       //read cooling water temperature and flow variables 
       //-------------------------------------------------
       IF NOT "SY".SIM_ON THEN                                                                                        // K01: Spare
           "DIS".ACT_WTR_FLW_XT_SFT   := INT_TO_REAL(WORD_TO_INT("P_BM_ACT_WTR_FLW_XT_SFT":P))/100.0;      // K02: seed shaft
           "DIS".ACT_WTR_TMP_XT_SFT   := INT_TO_REAL(WORD_TO_INT("P_BM_ACT_WTR_TMP_XT_SFT":P))/40.0;       
           "DIS".ACT_WTR_FLW_GCH      := INT_TO_REAL(WORD_TO_INT("P_BM_ACT_WTR_FLW_GCH":P))/100.0;         // K03: gate chamber 
           "DIS".ACT_WTR_TMP_GCH      := INT_TO_REAL(WORD_TO_INT("P_BM_ACT_WTR_TMP_GCH":P))/40.0; 
           "DIS".ACT_WTR_FLW_GCH_H    := INT_TO_REAL(WORD_TO_INT("P_BM_ACT_WTR_FLW_GCH_H":P))/100.0;       // K04: gate chamber valve housing
           "DIS".ACT_WTR_TMP_GCH_H    := INT_TO_REAL(WORD_TO_INT("P_BM_ACT_WTR_TMP_GCH_H":P))/40.0;    
           "DIS".ACT_WTR_FLW_GCH_V    := INT_TO_REAL(WORD_TO_INT("P_BM_ACT_WTR_FLW_GCH_V":P))/100.0;       // K05: gate chamber valve
           "DIS".ACT_WTR_TMP_GCH_V    := INT_TO_REAL(WORD_TO_INT("P_BM_ACT_WTR_TMP_GCH_V":P))/40.0;    
           "DIS".ACT_WTR_FLW_VPTS     := INT_TO_REAL(WORD_TO_INT("P_BM_ACT_WTR_FLW_VPTS":P))/100.0;        // K06: view ports
           "DIS".ACT_WTR_TMP_VPTS     := INT_TO_REAL(WORD_TO_INT("P_BM_ACT_WTR_TMP_VPTS":P))/40.0;    
           "DIS".ACT_WTR_FLW_TCH      := INT_TO_REAL(WORD_TO_INT("P_BM_ACT_WTR_FLW_TCH":P))/100.0;         // K07: top chamber 
           "DIS".ACT_WTR_TMP_TCH      := INT_TO_REAL(WORD_TO_INT("P_BM_ACT_WTR_TMP_TCH":P))/40.0;    
           "DIS".ACT_WTR_FLW_TEC_FLG  := INT_TO_REAL(WORD_TO_INT("P_BM_ACT_WTR_FLW_TEC_FLG":P))/100.0;     // K08: technology flange
           "DIS".ACT_WTR_TMP_TEC_FLG  := INT_TO_REAL(WORD_TO_INT("P_BM_ACT_WTR_TMP_TEC_FLG":P))/40.0;    
                                                                                                   // K09: Spare
           "DIS".ACT_WTR_FLW_UP_FCH   := INT_TO_REAL(WORD_TO_INT("P_BM_ACT_WTR_FLW_UP_FCH":P))/100.0;      // K10: Upper furnace chamber
           "DIS".ACT_WTR_TMP_UP_FCH   := INT_TO_REAL(WORD_TO_INT("P_BM_ACT_WTR_TMP_UP_FCH":P))/40.0;    
           "DIS".ACT_WTR_FLW_FCH      := INT_TO_REAL(WORD_TO_INT("P_BM_ACT_WTR_FLW_FCH":P))/100.0;         // K11: Lower furnace chamber
           "DIS".ACT_WTR_TMP_FCH      := INT_TO_REAL(WORD_TO_INT("P_BM_ACT_WTR_TMP_FCH":P))/40.0;    
           "DIS".ACT_WTR_FLW_VSL      := INT_TO_REAL(WORD_TO_INT("P_BM_ACT_WTR_FLW_BCH":P))/100.0;         // K12: bottom chamber
           "DIS".ACT_WTR_TMP_VSL      := INT_TO_REAL(WORD_TO_INT("P_BM_ACT_WTR_TMP_BCH":P))/40.0;    
           "DIS".ACT_WTR_FLW_SOC_BCH  := INT_TO_REAL(WORD_TO_INT("P_BM_ACT_WTR_FLW_SOC_BCH":P))/100.0;     // K13: socket bottom chamber
           "DIS".ACT_WTR_TMP_SOC_BCH  := INT_TO_REAL(WORD_TO_INT("P_BM_ACT_WTR_TMP_SOC_BCH":P))/40.0;    
           "DIS".ACT_WTR_FLW_CUR_FEED := INT_TO_REAL(WORD_TO_INT("P_BM_ACT_WTR_FLW_CFT_M":P))/100.0;       // K14: current feed throught Main
           "DIS".ACT_WTR_TMP_CUR_FEED := INT_TO_REAL(WORD_TO_INT("P_BM_ACT_WTR_TMP_CFT_M":P))/40.0;    
           "DIS".ACT_WTR_FLW_CFT_2    := INT_TO_REAL(WORD_TO_INT("P_BM_ACT_WTR_FLW_CFT_B":P))/100.0;       // K15: current feed throughs Bottom
           "DIS".ACT_WTR_TMP_CFT_2    := INT_TO_REAL(WORD_TO_INT("P_BM_ACT_WTR_TMP_CFT_B":P))/40.0;    
         //DIS.ACT_WTR_FLW_ACC      := INT_TO_REAL(WORD_TO_INT(BM_ACT_WTR_FLW_ACC))/100.0;        // K16: Active cooling
         //DIS.ACT_WTR_TMP_ACC      := INT_TO_REAL(WORD_TO_INT(BM_ACT_WTR_TMP_ACC))/40.0;   
           "DIS".ACT_WTR_FLW_CR_SFT   := INT_TO_REAL(WORD_TO_INT("P_BM_ACT_WTR_FLW_CR_SFT":P))/100.0;      // K17: crucible shaft
           "DIS".ACT_WTR_TMP_CR_SFT   := INT_TO_REAL(WORD_TO_INT("P_BM_ACT_WTR_TMP_CR_SFT":P))/40.0;    
           "DIS".ACT_WTR_FLW_PWR_CAB  := INT_TO_REAL(WORD_TO_INT("P_BM_ACT_WTR_FLW_PWR_CAB":P))/100.0;     // K18: high current cables Main
           "DIS".ACT_WTR_TMP_PWR_CAB  := INT_TO_REAL(WORD_TO_INT("P_BM_ACT_WTR_TMP_PWR_CAB":P))/40.0;    
           "DIS".ACT_WTR_FLW_PWR_CAB2 := INT_TO_REAL(WORD_TO_INT("P_BM_ACT_WTR_FLW_PWR_CAB2":P))/100.0;    // K19: high current cables Bot
           "DIS".ACT_WTR_TMP_PWR_CAB2 := INT_TO_REAL(WORD_TO_INT("P_BM_ACT_WTR_TMP_PWR_CAB2":P))/40.0;    
           "DIS".ACT_WTR_FLW_HTR_1    := INT_TO_REAL(WORD_TO_INT("P_BM_ACT_WTR_FLW_HTR":P))/100.0;         // K20: heater power supply
           "DIS".ACT_WTR_TMP_HTR_1    := INT_TO_REAL(WORD_TO_INT("P_BM_ACT_WTR_TMP_HTR":P))/40.0;         
                                                                                                   // K21: Spare
                                                                                                   // K22: Spare
                                                                                                   // K23: Spare
           "DIS".ACT_WTR_FLW_GCH_ADDS      := INT_TO_REAL(WORD_TO_INT("P_BM_ACT_WTR_FLW_GCH_ADDS":P))/100.0;         // K24: gate chamber Additions
           "DIS".ACT_WTR_TMP_GCH_ADDS      := INT_TO_REAL(WORD_TO_INT(SHR(IN:= "P_BM_ACT_WTR_TMP_GCH_ADDS":P, N:= 2)))/10.0;    
         //DIS.ACT_WTR_FLW_PU       := INT_TO_REAL(WORD_TO_INT(BM_ACT_WTR_FLW_PU))/100.0;          // K25: pump unit
         //DIS.ACT_WTR_TMP_PU       := INT_TO_REAL(WORD_TO_INT(SHR(IN:= BM_ACT_WTR_TMP_PU, N:= 2)))/10.0;    
           "DIS".ACT_WTR_FLW_MAG_CO4  := INT_TO_REAL(WORD_TO_INT("P_BM_ACT_WTR_FLW_MAG_CO4":P))/100.0;     // K26: magnet compressor unit 4
           "DIS".ACT_WTR_TMP_MAG_CO4  := INT_TO_REAL(WORD_TO_INT(SHR(IN:= "P_BM_ACT_WTR_TMP_MAG_CO4":P, N:= 2)))/10.0;    
           "DIS".ACT_WTR_FLW_MAG_CO3  := INT_TO_REAL(WORD_TO_INT("P_BM_ACT_WTR_FLW_MAG_CO3":P))/100.0;     // K27: magnet compressor unit 3
           "DIS".ACT_WTR_TMP_MAG_CO3  := INT_TO_REAL(WORD_TO_INT(SHR(IN:= "P_BM_ACT_WTR_TMP_MAG_CO3":P, N:= 2)))/10.0;    
           "DIS".ACT_WTR_FLW_MAG_CO2  := INT_TO_REAL(WORD_TO_INT("P_BM_ACT_WTR_FLW_MAG_CO2":P))/100.0;     // K28: magnet compressor unit 2
           "DIS".ACT_WTR_TMP_MAG_CO2  := INT_TO_REAL(WORD_TO_INT(SHR(IN:= "P_BM_ACT_WTR_TMP_MAG_CO2":P, N:= 2)))/10.0;    
           "DIS".ACT_WTR_FLW_MAG_CO1  := INT_TO_REAL(WORD_TO_INT("P_BM_ACT_WTR_FLW_MAG_CO1":P))/100.0;     // K29: magnet compressor unit 1
           "DIS".ACT_WTR_TMP_MAG_CO1  := INT_TO_REAL(WORD_TO_INT(SHR(IN:= "P_BM_ACT_WTR_TMP_MAG_CO1":P, N:= 2)))/10.0;    
           "DIS".ACT_WTR_FLW_MAG_CAB  := INT_TO_REAL(WORD_TO_INT("P_BM_ACT_WTR_FLW_MAG_CAB":P))/100.0;     // K30: magnet power supply
           "DIS".ACT_WTR_TMP_MAG_CAB  := INT_TO_REAL(WORD_TO_INT(SHR(IN:= "P_BM_ACT_WTR_TMP_MAG_CAB":P, N:= 2)))/10.0;    

           "DIS".ACT_WTR_FLW_VAC_BYP  := INT_TO_REAL(WORD_TO_INT("P_BM_ACT_WTR_FLW_VAC_BYP":P))/100.0;     // Kxx: vacuum bypass tube
           "DIS".ACT_WTR_TMP_VAC_BYP  := INT_TO_REAL(WORD_TO_INT("P_BM_ACT_WTR_TMP_VAC_BYP":P))/40.0;  
       END_IF;


       //set water flow and temperature alarms
       //-------------------------------------
       "FLT".XT_TAS              :=  ("DIS".ACT_WTR_TMP_XT_SFT > "CNF".WTR_TMP_WRN);             // seed shaft
       "FLT".XT_WFS              :=  ("DIS".ACT_WTR_FLW_XT_SFT < "CNF".MIN_WTR_FLW_XT_SFT);       
       "FLT".WTR_TMP_GCH         :=  ("DIS".ACT_WTR_TMP_GCH > "CNF".WTR_TMP_WRN) OR              //gate chamber
                                   ("DIS".ACT_WTR_TMP_GCH_H > "CNF".WTR_TMP_WRN);              // gate chamber valve housing    
       "FLT".WTR_FLW_GCH         :=  ("DIS".ACT_WTR_FLW_GCH < "CNF".MIN_WTR_FLW_GCH) OR 
                                   ("DIS".ACT_WTR_FLW_GCH_H < "CNF".MIN_WTR_FLW_GCH_H);  
       "FLT".WTR_TMP_GCH_V       :=  ("DIS".ACT_WTR_TMP_GCH_V > "CNF".WTR_TMP_WRN);              //gate chamber valve
       "FLT".WTR_FLW_GCH_V       :=  ("DIS".ACT_WTR_FLW_GCH_V < "CNF".MIN_WTR_FLW_GCH_V); 
       "FLT".WTR_TMP_VPTS        :=  ("DIS".ACT_WTR_TMP_VPTS > "CNF".WTR_TMP_WRN);               //view ports
       "FLT".WTR_FLW_VPTS        :=  ("DIS".ACT_WTR_FLW_VPTS < "CNF".MIN_WTR_FLW_VPTS); 
       "FLT".WTR_TMP_TCH         :=  ("DIS".ACT_WTR_TMP_TCH > "CNF".WTR_TMP_WRN);                //top chamber
       "FLT".WTR_FLW_TCH         :=  ("DIS".ACT_WTR_FLW_TCH < "CNF".MIN_WTR_FLW_TCH);
       "FLT".WTR_TMP_TEC_FLG     :=  ("DIS".ACT_WTR_TMP_TEC_FLG > "CNF".WTR_TMP_WRN);            //technology flange
       "FLT".WTR_FLW_TEC_FLG     :=  ("DIS".ACT_WTR_FLW_TEC_FLG < "CNF".MIN_WTR_FLW_TEC_CHB);    
       "FLT".WTR_TMP_FCH         :=  ("DIS".ACT_WTR_TMP_UP_FCH > "CNF".WTR_TMP_WRN)OR            //upper furnace chamber
                                   ("DIS".ACT_WTR_TMP_FCH > "CNF".WTR_TMP_WRN);                //lower furnace chamber
       "FLT".WTR_FLW_FCH         :=  ("DIS".ACT_WTR_FLW_UP_FCH < "CNF".MIN_WTR_FLW_FCH)OR
                                   ("DIS".ACT_WTR_FLW_FCH < "CNF".MIN_WTR_FLW_FCH);
       "FLT".WTR_TMP_VSL         :=  ("DIS".ACT_WTR_TMP_VSL  > "CNF".WTR_TMP_WRN) OR             //bottom chamber
                                   ("DIS".ACT_WTR_TMP_SOC_BCH > "CNF".WTR_TMP_WRN);            //socket bottom chamber    
       "FLT".WTR_FLW_VSL         :=  ("DIS".ACT_WTR_FLW_VSL < "CNF".MIN_WTR_FLW_VSL) OR
                                   ("DIS".ACT_WTR_FLW_SOC_BCH < "CNF".MIN_WTR_FLW_VSL);    
       "FLT".WTR_TMP_CUR_FEED    :=  ("DIS".ACT_WTR_TMP_CUR_FEED > "CNF".WTR_TMP_WRN);           //current feed throughs heater 1
       "FLT".WTR_FLW_CUR_FEED    :=  ("DIS".ACT_WTR_FLW_CUR_FEED < "CNF".MIN_WTR_FLW_CUR_FEED); 
       "FLT".WTR_TMP_CFT_2       :=  ("DIS".ACT_WTR_TMP_CFT_2 > "CNF".WTR_TMP_WRN);              //current feed throughs heater 2
       "FLT".WTR_FLW_CFT_2       :=  ("DIS".ACT_WTR_FLW_CFT_2 < "CNF".MIN_WTR_FLW_CUR_FEED);
       "FLT".WTR_TMP_PWR_CAB     :=  ("DIS".ACT_WTR_TMP_PWR_CAB > "CNF".WTR_TMP_WRN)OR           //high current cables main
                                   ("DIS".ACT_WTR_TMP_PWR_CAB2 > "CNF".WTR_TMP_WRN);           //high current cables 2 bot    
       "FLT".WTR_FLW_PWR_CAB     :=  ("DIS".ACT_WTR_FLW_PWR_CAB < "CNF".MIN_WTR_FLW_PWR_CAB)OR 
                                   ("DIS".ACT_WTR_FLW_PWR_CAB2 < "CNF".MIN_WTR_FLW_PWR_CAB); 
       "FLT".WTR_TMP_CR_SFT      :=  ("DIS".ACT_WTR_TMP_CR_SFT > "CNF".WTR_TMP_WRN);             //crucible shaft
       "FLT".WTR_FLW_CR_SFT      :=  ("DIS".ACT_WTR_FLW_CR_SFT < "CNF".MIN_WTR_FLW_CR_SFT);    
       "FLT".WTR_TMP_HTR_1       :=  ("DIS".ACT_WTR_TMP_HTR_1 > "CNF".WTR_TMP_WRN);              //heater power supply
       IF "CNF".CONF_PWR_SPL_TYPE = 1 THEN 
          "FLT".WTR_FLW_HTR_1       :=  ("DIS".ACT_WTR_FLW_HTR_1 < "CNF".MIN_WTR_FLW_PWR_HTR_1); 
       END_IF;
       IF "CNF".CONF_PWR_SPL_TYPE = 2 THEN 
          "FLT".WTR_FLW_HTR_1       :=  ("DIS".ACT_WTR_FLW_HTR_1 < "CNF".MIN_WTR_FLW_INJ_HTR_1); 
       END_IF;
     //FLT.WTR_TMP_ACC         :=  (DIS.ACT_WTR_TMP_ACC > CNF.WTR_TMP_WRN);                 // active cooling
     //FLT.WTR_FLW_ACC         :=  (DIS.ACT_WTR_FLW_ACC < CNF.MIN_WTR_FLW_ACC_IN);         
       "FLT".WTR_TMP_GCH_ADDS         :=  ("DIS".ACT_WTR_TMP_GCH_ADDS > "CNF".WTR_TMP_WRN);                 // chamber parts, view ports
       "FLT".WTR_FLW_GCH_ADDS         :=  ("DIS".ACT_WTR_FLW_GCH_ADDS < "CNF".MIN_WTR_FLW_GCH_ADDS);    

       "FLT".MAG_TAS             :=  ("DIS".ACT_WTR_TMP_MAG_CO1 > "CNF".WTR_TMP_WRN) OR           // magnet compressor unit 1
                                   ("DIS".ACT_WTR_TMP_MAG_CO2 > "CNF".WTR_TMP_WRN) OR           // magnet compressor unit 2
                                   ("DIS".ACT_WTR_TMP_MAG_CO3 > "CNF".WTR_TMP_WRN) OR           // magnet compressor unit 3
                                   ("DIS".ACT_WTR_TMP_MAG_CO4 > "CNF".WTR_TMP_WRN) OR           // magnet compressor unit 4
                                   ("DIS".ACT_WTR_TMP_MAG_CAB > "CNF".WTR_TMP_WRN);             // magnet power supply
       "FLT".MAG_WFS             :=  ("DIS".ACT_WTR_FLW_MAG_CO1 < "CNF".MIN_WTR_FLW_MAG_COMP) OR    
                                   ("DIS".ACT_WTR_FLW_MAG_CO2 < "CNF".MIN_WTR_FLW_MAG_COMP) OR    
                                   ("DIS".ACT_WTR_FLW_MAG_CO3 < "CNF".MIN_WTR_FLW_MAG_COMP) OR    
                                   ("DIS".ACT_WTR_FLW_MAG_CO4 < "CNF".MIN_WTR_FLW_MAG_COMP) OR    
                                   ("DIS".ACT_WTR_FLW_MAG_CAB < "CNF".MIN_WTR_FLW_MAG_CAB);    

       "FLT".WTR_TMP_VAC_BYP     :=  ("DIS".ACT_WTR_TMP_VAC_BYP > "CNF".WTR_TMP_WRN);                // vacuum bypass tube - not included in interlocks
       "FLT".WTR_FLW_VAC_BYP     :=  ("DIS".ACT_WTR_FLW_VAC_BYP < "CNF".MIN_WTR_FLW_VAC_BYP);

       //built shut down flag low water flow (current feed throughs heater 2 not included)
       //---------------------------------------------------------------------------------
       #low_wtr_flw :=      "FLT".XT_WFS OR                   //seed shaft
                           "FLT".WTR_FLW_GCH OR              //gate chamber or gate chamber valve housing
                           "FLT".WTR_FLW_GCH_V OR            //gate chamber valve
                           "FLT".WTR_FLW_VPTS OR             //view ports
                           "FLT".WTR_FLW_TCH OR              //top chamber
                           "FLT".WTR_FLW_TEC_FLG OR          //technology flange
                           "FLT".WTR_FLW_FCH OR              //upper furnace chamber or lower furnace chamber
                           "FLT".WTR_FLW_VSL OR              //bottom chamber or socket bottom chamber
                           "FLT".WTR_FLW_CR_SFT OR           //crucible shaft
                           "FLT".WTR_FLW_HTR_1 OR            //heater power supply
                           "FLT".WTR_FLW_GCH_ADDS;           //gate chamber additions

       //built shut down flag low water flow heater 1(only current feed throughs and cables of heater 1)
       //-----------------------------------------------------------------------------------------------
       #low_wtr_flw_htr_1   :=  ("DIS".ACT_WTR_FLW_CUR_FEED < "CNF".MIN_WTR_FLW_CUR_FEED) OR        //current feed throughs heater 1
                               "DIS".ACT_WTR_FLW_PWR_CAB < "CNF".MIN_WTR_FLW_PWR_CAB;             //high current cables heater 1

       //built shut down flag low water flow heater 2(only current feed throughs and cables of heater 2)
       //-----------------------------------------------------------------------------------------------
       #low_wtr_flw_htr_2   :=  ("DIS".ACT_WTR_FLW_CFT_2 < "CNF".MIN_WTR_FLW_CUR_FEED) OR           //current feed throughs heater 2
                               "DIS".ACT_WTR_FLW_PWR_CAB2 < "CNF".MIN_WTR_FLW_PWR_CAB;             //high current cables heater 2

       //built shut down flag high water temperature (current feed throughs heater 2 not included)
       //-----------------------------------------------------------------------------------------
       #high_wtr_tmp    :=  ("DIS".ACT_WTR_TMP_XT_SFT > "CNF".MAX_WTR_TMP_LIM)OR    //seed shaft
                           ("DIS".ACT_WTR_TMP_GCH > "CNF".MAX_WTR_TMP_LIM) OR      //gate chamber
                           ("DIS".ACT_WTR_TMP_GCH_H > "CNF".MAX_WTR_TMP_LIM)OR     //gate chamber valve housing    
                           ("DIS".ACT_WTR_TMP_GCH_V > "CNF".MAX_WTR_TMP_LIM)OR     //gate chamber valve
                           ("DIS".ACT_WTR_TMP_VPTS > "CNF".MAX_WTR_TMP_LIM)OR      //view ports
                           ("DIS".ACT_WTR_TMP_TCH > "CNF".MAX_WTR_TMP_LIM)OR       //top chamber
                           ("DIS".ACT_WTR_TMP_TEC_FLG > "CNF".MAX_WTR_TMP_LIM)OR   //technology flange
                           ("DIS".ACT_WTR_TMP_UP_FCH > "CNF".MAX_WTR_TMP_LIM)OR    //upper furnace chamber
                           ("DIS".ACT_WTR_TMP_FCH > "CNF".MAX_WTR_TMP_LIM)OR       //lower furnace chamber
                           ("DIS".ACT_WTR_TMP_VSL  > "CNF".MAX_WTR_TMP_LIM) OR     //bottom chamber
                           ("DIS".ACT_WTR_TMP_SOC_BCH > "CNF".MAX_WTR_TMP_LIM)OR   //socket bottom chamber    
                           ("DIS".ACT_WTR_TMP_CR_SFT > "CNF".MAX_WTR_TMP_LIM)OR    //crucible shaft
                           ("DIS".ACT_WTR_TMP_HTR_1 > "CNF".MAX_WTR_TMP_LIM)OR     //heater power supply
                           ("DIS".ACT_WTR_TMP_GCH_ADDS > "CNF".MAX_WTR_TMP_LIM);   //gate chamber additions

       "FLT".WTR_TMP_VAC_BYP     :=  ("DIS".ACT_WTR_TMP_VAC_BYP > "CNF".WTR_TMP_WRN);                // vacuum bypass tube - not included in interlocks
       "FLT".WTR_FLW_VAC_BYP     :=  ("DIS".ACT_WTR_FLW_VAC_BYP < "CNF".MIN_WTR_FLW_VAC_BYP);

       //built shut down flag high cooling water temperature heater 1
       //------------------------------------------------------------
       #high_wtr_tmp_htr_1  :=  ("DIS".ACT_WTR_TMP_CUR_FEED > "CNF".MAX_WTR_TMP_LIM) OR //current feed throughs heater 1
                               ("DIS".ACT_WTR_TMP_PWR_CAB > "CNF".MAX_WTR_TMP_LIM);    //high current cables heater 1

       //built shut down flag high cooling water temperature heater 2
       //------------------------------------------------------------
       #high_wtr_tmp_htr_2  :=  ("DIS".ACT_WTR_TMP_CFT_2 > "CNF".MAX_WTR_TMP_LIM) OR    //current feed throughs heater 2
                               ("DIS".ACT_WTR_TMP_PWR_CAB2 > "CNF".MAX_WTR_TMP_LIM);   //high current cables heater 2

       //set alarm high water temperature
       //--------------------------------            
       "FLT".WTR_TMP_HIGH_LIM    :=  #high_wtr_tmp OR            
                                   #high_wtr_tmp_htr_1 OR
                                   #high_wtr_tmp_htr_2;

       //reconnect heater 1 after power fail
       //-----------------------------------
       IF "DV".PWR_FAIL_HTR_1_ON THEN
           "KYA".SET_HTR_1_PWR := "AV".PWR_FAIL_HTR_1_PWR;      // restore last power value

           IF ("LT".HTR_1_ON) THEN  //AND PDO.HTR_1_ENB
               "DV".PWR_FAIL_HTR_1_ON := false;               // delete request, if heater on
               "AV".PWR_FAIL_HTR_1_PWR := 0.0;
           END_IF;
       END_IF;

       //check heater power supply interlocks affecting all heater
       //---------------------------------------------------------
       #htr_itl_ok      :=  "BM_HTR_ITL" (aps             :=      NOT "PDI".FCH_APS,  
                                       tas             :=      NOT #high_wtr_tmp,
                                       on_dly_tas      :=      "HTR_TAS_DLY", 
                                       dly_time_tas    :=      T#30s,
                                       wfs             :=      NOT #low_wtr_flw,
                                       on_dly_wfs      :=      "HTR_WFS_DLY", 
                                       dly_time_wfs    :=      T#30s,                                               
                                       aux             :=      "DV".MAIN_SWITCH_ON AND
                                                              ("PDI".ACC_SC_HTR_OK AND   //ACC heater safety circuit
                                                               "PDI".ACC_SC_WTR_OK OR    //ACC water safety circuit
                                                               NOT "DV".ACC_INST),           //ACC installed?
                                       on_dly_aux      :=      "HTR_AUX_DLY", 
                                       dly_time_aux    :=      T#1s);  

       //extend reset flag earth fault detection
       //---------------------------------------   
       "LT".RESET_ERR_HTR_ETH    := "SysOffdelay" (DIN     := "KYD".RESET_ERR_HTR_ETH,
                                               SetTime := 20,                          // setp. time
                                               ActTime := #rst_err_htr_eth_dly,         // act. time
                                               Tick    := "SysTick100ms");               // timebase (100ms)


       //TLU switching power supply
       //--------------------------
       //check heater 1 interlock
       //------------------------
       #htr_1_itl_ok    :=  "BM_HTR_ITL" (aps             :=      true,  
                                       tas             :=      NOT #high_wtr_tmp_htr_1,
                                       on_dly_tas      :=      "HTR_1_TAS_DLY", 
                                       dly_time_tas    :=      T#30s,
                                       wfs             :=      NOT #low_wtr_flw_htr_1,
                                       on_dly_wfs      :=      "HTR_1_WFS_DLY", 
                                       dly_time_wfs    :=      T#30s,                                               
                                       aux             :=      NOT "FLT".HTR_1_PWR_SPL,
                                       on_dly_aux      :=      "HTR_1_AUX_DLY", 
                                       dly_time_aux    :=      T#1s);                                

       //check heater 2 interlock
       //------------------------
       #htr_2_itl_ok    :=  "BM_HTR_ITL" (aps             :=      true,  
                                       tas             :=      NOT #high_wtr_tmp_htr_2,
                                       on_dly_tas      :=      "HTR_2_TAS_DLY", 
                                       dly_time_tas    :=      T#30s,
                                       wfs             :=      NOT #low_wtr_flw_htr_2,
                                       on_dly_wfs      :=      "HTR_2_WFS_DLY", 
                                       dly_time_wfs    :=      T#30s,                                               
                                       aux             :=      NOT "FLT".HTR_2_PWR_SPL,
                                       on_dly_aux      :=      "HTR_2_AUX_DLY", 
                                       dly_time_aux    :=      T#1s);                                

       //call control module of heater 1
       //-------------------------------
       "CM_ITL_IO"(ADR := 30,
              KYD_ON := ("KYD".HTR_1_ON AND NOT "DV".EMG_DRV_ENB) OR "DV".PWR_FAIL_HTR_1_ON,
              KYD_OFF:= "KYD".HTR_1_OFF OR "DV".PWR_FAIL_HTR_OFF OR "DV".EMG_DVC_OFF,
              AUTO := "APC".AUTOMATIC,
              DC_ON:= "DC".HTR_1_ON,
              CON1 := "PDI".EMO,
              CON2 := "DV".MAIN_SWITCH_ON,
              CON3 := #htr_itl_ok,
              CON4 := #htr_1_itl_ok,               
              CON5 := "SysLog1",
              CON6 := "SysLog1",                             
              CON7 := "SysLog1",                             
              CON8 := "SysLog1",
              ITL_OUT:= "STA_ITL_CAUSE",
              LT_OUT := "LT".HTR_1_ON);

       //set power enable delayed
       //------------------------
       #htr_1_enb     := "SysOndelay"(DIN     := "LT".HTR_1_ON,
                                   SetTime := 10,                // 1 sec. delay after power on
                                   ActTime := #htr_1_pwr_enb_dly, // act. time
                                   Tick    := "SysTick100ms");     // timebase (100ms)

       //heater supply power on
       //----------------------
       "PDO".HTR_PWR_ON    :=  "LT".HTR_1_ON;               

       //reset power set point if heater enable is gone
       //----------------------------------------------
       IF NOT #htr_1_enb  THEN
           "KYA".SET_HTR_1_PWR  := 0.0;
           "CTL".SET_HTR_1_PWR  := 0.0;
       END_IF;

       //extent reset flag
       //-----------------
       "LT".RST_HTR_1_PWR_SPL := "SysOffdelay"(DIN     := "KYD".RST_HTR_1_PWR_SPL,
                                           SetTime := 20,                          // setp. time
                                           ActTime := #rst_htr_1_pwr_spl_dly,       // act. time
                                           Tick    := "SysTick100ms");               // timebase (100ms)

       //call control module of heater 2
       //-------------------------------
       "CM_ITL_IO"(ADR := 31,
              KYD_ON := ("KYD".HTR_2_ON AND NOT "DV".EMG_DRV_ENB) OR "DV".PWR_FAIL_HTR_2_ON,
              KYD_OFF:= "KYD".HTR_2_OFF OR "DV".PWR_FAIL_HTR_OFF OR "DV".EMG_DVC_OFF,
              AUTO := "APC".AUTOMATIC,
              DC_ON:= "DC".HTR_2_ON,
              CON1 := "PDI".EMO,
              CON2 := "DV".MAIN_SWITCH_ON,
              CON3 := #htr_itl_ok,
              CON4 := #htr_2_itl_ok,               
              CON5 := "SysLog1",
              CON6 := "SysLog1",                             
              CON7 := "SysLog1",                             
              CON8 := "SysLog1",
              ITL_OUT:= "STA_ITL_CAUSE",
              LT_OUT := "LT".HTR_2_ON);

       //set power enable delayed
       //------------------------
       #htr_2_enb     := "SysOndelay"(DIN     := "LT".HTR_2_ON,
                                   SetTime := 10,                // 1 sec. delay after power on
                                   ActTime := #htr_2_pwr_enb_dly, // act. time
                                   Tick    := "SysTick100ms");     // timebase (100ms)

       //set output heater 2 (used in ekz_sm_pwr_fail)
       //---------------------------------------------
      // PDO.HTR_2_ON    :=  LT.HTR_2_ON;               

       //reset power set point if heater enable is gone
       //----------------------------------------------
       IF NOT #htr_2_enb  THEN
           "KYA".SET_HTR_2_PWR  := 0.0;
           "CTL".SET_HTR_2_PWR  := 0.0;
       END_IF;

       //extent reset flag
       //-----------------
       "LT".RST_HTR_2_PWR_SPL := "SysOffdelay"(DIN     := "KYD".RST_HTR_2_PWR_SPL,
                                           SetTime := 20,                          // setp. time
                                           ActTime := #rst_htr_2_pwr_spl_dly,       // act. time
                                           Tick    := "SysTick100ms");               // timebase (100ms)


       //call communication module with TLU profibus interface
       //-----------------------------------------------------
       IF "CNF".CONF_PWR_SPL_TYPE = 1 THEN    
           //delay communication 
           //-------------------
           #start_htr_com := "SysOndelay"(DIN     := "PDO".HTR_PWR_ON,
                                       SetTime := 30,                  // setp. time
                                       ActTime := #com_heater_dly,      // act. time
                                       Tick    := "SysTick100ms");

           IF #start_htr_com THEN 

               #PM_TLU_HTR_1(   htr_enb         :=  #htr_1_enb, 
                               htr_rst         :=  "LT".RST_HTR_1_PWR_SPL,
                               fst_byte_offs   :=  0,        
                               dp_adress       :=  16#380,                 //addr: 896      
                               set_htr_pwr     :=  "CTL".SET_HTR_1_PWR,
                               htr_pwr_rng     :=  "CNF".HTR_1_PWR_RANGE,
                               htr_cur_rng     :=  "CNF".HTR_1_CUR_RANGE,
                               htr_vlt_rng     :=  "CNF".HTR_1_VLT_RANGE);
           END_IF;                

           "AV".ACT_HTR_1_PWR        :=  #PM_TLU_HTR_1.act_htr_pwr; 
           "AV".ACT_HTR_1_CUR        :=  #PM_TLU_HTR_1.act_htr_cur; 
           "AV".ACT_HTR_1_VLT        :=  #PM_TLU_HTR_1.act_htr_vlt; 

           "FLT".HTR_1_PWR_SPL_WRN   :=  #PM_TLU_HTR_1.sta_warn;  
           "FLT".HTR_1_PWR_SPL       :=  #PM_TLU_HTR_1.sta_error;  

           #htr_1_is_on             :=  #PM_TLU_HTR_1.sta_htr_on;         
           #htr_1_pi_mode           :=  #PM_TLU_HTR_1.sta_pi_mode;     
           #htr_1_pu_mode           :=  #PM_TLU_HTR_1.sta_pu_mode;      
           #htr_1_i_mode            :=  #PM_TLU_HTR_1.sta_i_mode;       
           #htr_1_u_mode            :=  #PM_TLU_HTR_1.sta_u_mode;       
           #htr_1_sta_saved         :=  #PM_TLU_HTR_1.sta_saved;         
           #htr_1_flt_i_pri         :=  #PM_TLU_HTR_1.flt_i_pri;       
           #htr_1_flt_i_max         :=  #PM_TLU_HTR_1.flt_i_max;        
           #htr_1_flt_u_max         :=  #PM_TLU_HTR_1.flt_u_max;        
           #htr_1_flt_wire          :=  #PM_TLU_HTR_1.flt_wire;           
           #htr_1_flt_flash         :=  #PM_TLU_HTR_1.flt_flash;          
           #htr_1_flt_trafo         :=  #PM_TLU_HTR_1.flt_trafo;         
           #htr_1_flt_data_flow     :=  #PM_TLU_HTR_1.flt_data_flow;    
           #htr_1_flt_data_com      :=  #PM_TLU_HTR_1.flt_data_com;      
           #htr_1_flt_data          :=  #PM_TLU_HTR_1.flt_data;       
           #htr_1_flt_tast          :=  #PM_TLU_HTR_1.flt_tast;            
           #htr_1_flt_ua_max        :=  #PM_TLU_HTR_1.flt_ua_max;          
           #htr_1_flt_u_min         :=  #PM_TLU_HTR_1.flt_u_min;          
           #htr_1_flt_temp          :=  #PM_TLU_HTR_1.flt_temp;            
           #htr_1_flt_sense         :=  #PM_TLU_HTR_1.flt_sense;         
           #htr_1_flt_igbt          :=  #PM_TLU_HTR_1.flt_igbt;          
           #htr_1_flt_dioden        :=  #PM_TLU_HTR_1.flt_dioden;       
           #htr_1_flt_3             :=  #PM_TLU_HTR_1.flt_3;             
           #htr_1_flt_shunt         :=  #PM_TLU_HTR_1.flt_shunt;         
           #htr_1_flt_board         :=  #PM_TLU_HTR_1.flt_board;         
           #htr_1_flt_6             :=  #PM_TLU_HTR_1.flt_6;            
           #htr_1_flt_soft          :=  #PM_TLU_HTR_1.flt_soft;          
           #htr_1_flt_timeout       :=  #PM_TLU_HTR_1.flt_timeout;        
           #htr_1_flt_short         :=  #PM_TLU_HTR_1.flt_short;    

           //errors heater 1 earthing monitoring
           //------------------ 
           IF  (("P_BM_HTR_1_ETH_STA":P AND 2#0001_0000) = 2#0001_0000) THEN  
               #flt_htr_1_eth_range := true;     //range error
           ELSE     
               #flt_htr_1_eth_range := false;
           END_IF;

           IF (("P_BM_HTR_1_ETH_STA":P AND 2#0010_0000) = 2#0010_0000) THEN 
               #flt_htr_1_eth_hw := true;       //intern hardware error
           ELSE     
               #flt_htr_1_eth_hw := false;
           END_IF;

           IF (("P_BM_HTR_1_ETH_STA":P AND 2#0100000) = 2#0100_0000) THEN 
               #flt_htr_1_eth_bus := true;      //bus error
           ELSE     
               #flt_htr_1_eth_bus := false;
           END_IF;

           //heater 2
           //--------  
           IF #start_htr_com THEN 

               #PM_TLU_HTR_2(   htr_enb         :=  #htr_2_enb, 
                               htr_rst         :=  "LT".RST_HTR_2_PWR_SPL,
                               fst_byte_offs   :=  0,        
                               dp_adress       :=  16#3C0,                 //addr: 960      
                               set_htr_pwr     :=  "CTL".SET_HTR_2_PWR,
                               htr_pwr_rng     :=  "CNF".HTR_2_PWR_RANGE,
                               htr_cur_rng     :=  "CNF".HTR_2_CUR_RANGE,
                               htr_vlt_rng     :=  "CNF".HTR_2_VLT_RANGE);
           END_IF;                

           "AV".ACT_HTR_2_PWR        :=  #PM_TLU_HTR_2.act_htr_pwr; 
           "AV".ACT_HTR_2_CUR        :=  #PM_TLU_HTR_2.act_htr_cur; 
           "AV".ACT_HTR_2_VLT        :=  #PM_TLU_HTR_2.act_htr_vlt; 

           "FLT".HTR_2_PWR_SPL_WRN   :=  #PM_TLU_HTR_2.sta_warn;  
           "FLT".HTR_2_PWR_SPL       :=  #PM_TLU_HTR_2.sta_error;    

           #htr_2_is_on             :=  #PM_TLU_HTR_2.sta_htr_on;         
           #htr_2_pi_mode           :=  #PM_TLU_HTR_2.sta_pi_mode;     
           #htr_2_pu_mode           :=  #PM_TLU_HTR_2.sta_pu_mode;      
           #htr_2_i_mode            :=  #PM_TLU_HTR_2.sta_i_mode;       
           #htr_2_u_mode            :=  #PM_TLU_HTR_2.sta_u_mode;       
           #htr_2_sta_saved         :=  #PM_TLU_HTR_2.sta_saved;         
           #htr_2_flt_i_pri         :=  #PM_TLU_HTR_2.flt_i_pri;       
           #htr_2_flt_i_max         :=  #PM_TLU_HTR_2.flt_i_max;        
           #htr_2_flt_u_max         :=  #PM_TLU_HTR_2.flt_u_max;        
           #htr_2_flt_wire          :=  #PM_TLU_HTR_2.flt_wire;           
           #htr_2_flt_flash         :=  #PM_TLU_HTR_2.flt_flash;          
           #htr_2_flt_trafo         :=  #PM_TLU_HTR_2.flt_trafo;         
           #htr_2_flt_data_flow     :=  #PM_TLU_HTR_2.flt_data_flow;    
           #htr_2_flt_data_com      :=  #PM_TLU_HTR_2.flt_data_com;      
           #htr_2_flt_data          :=  #PM_TLU_HTR_2.flt_data;       
           #htr_2_flt_tast          :=  #PM_TLU_HTR_2.flt_tast;            
           #htr_2_flt_ua_max        :=  #PM_TLU_HTR_2.flt_ua_max;          
           #htr_2_flt_u_min         :=  #PM_TLU_HTR_2.flt_u_min;          
           #htr_2_flt_temp          :=  #PM_TLU_HTR_2.flt_temp;            
           #htr_2_flt_sense         :=  #PM_TLU_HTR_2.flt_sense;         
           #htr_2_flt_igbt          :=  #PM_TLU_HTR_2.flt_igbt;          
           #htr_2_flt_dioden        :=  #PM_TLU_HTR_2.flt_dioden;       
           #htr_2_flt_3             :=  #PM_TLU_HTR_2.flt_3;             
           #htr_2_flt_shunt         :=  #PM_TLU_HTR_2.flt_shunt;         
           #htr_2_flt_board         :=  #PM_TLU_HTR_2.flt_board;         
           #htr_2_flt_6             :=  #PM_TLU_HTR_2.flt_6;            
           #htr_2_flt_soft          :=  #PM_TLU_HTR_2.flt_soft;          
           #htr_2_flt_timeout       :=  #PM_TLU_HTR_2.flt_timeout;        
           #htr_2_flt_short         :=  #PM_TLU_HTR_2.flt_short;  

           //errors heater 2 earthing monitoring
           //------------------ 
           IF  (("P_BM_HTR_2_ETH_STA":P AND 2#0001_0000) = 2#0001_0000) THEN  
               #flt_htr_2_eth_range := true;    //range error
           ELSE     
               #flt_htr_2_eth_range := false;
           END_IF;

           IF (("P_BM_HTR_2_ETH_STA":P AND 2#0010_0000) = 2#0010_0000) THEN 
               #flt_htr_2_eth_hw := true;       //intern hardware error
           ELSE     
               #flt_htr_2_eth_hw := false;
           END_IF;

           IF (("P_BM_HTR_2_ETH_STA":P AND 2#0100000) = 2#0100_0000) THEN 
               #flt_htr_2_eth_bus := true;      //bus error
           ELSE     
               #flt_htr_2_eth_bus := false;
           END_IF;

           // heater earthing monitoring error on HMI
           //------------------
           "FLT".HTR_ERH_COMM :=   #flt_htr_1_eth_range 
                              OR #flt_htr_1_eth_hw 
                              OR #flt_htr_1_eth_bus 
                              OR #flt_htr_2_eth_range
                              OR #flt_htr_2_eth_hw
                              OR #flt_htr_2_eth_bus;

           // reset heater earthing monitoring errors
           //------------------ 
           IF  "LT".RESET_ERR_HTR_ETH THEN 
               "P_BM_HTR_1_ETH_CTRL":P := 2#0100_0000;
               "P_BM_HTR_2_ETH_CTRL":P := 2#0100_0000;
           ELSE
               "P_BM_HTR_1_ETH_CTRL":P := 2#0000_0000;
               "P_BM_HTR_2_ETH_CTRL":P := 2#0000_0000;
           END_IF;

       END_IF;

       IF "CNF".CONF_PWR_SPL_TYPE = 2 THEN
           //call communication module with Injet profinet interface
           //-----------------------------------------------------
           //call Injet function  
           #PM_INJET_HTR     (htr_1_enb     := #htr_1_enb,  
                             htr_2_enb     := #htr_2_enb,     
                             set_htr_1_pwr := "CTL".SET_HTR_1_PWR,
                             set_htr_2_pwr := "CTL".SET_HTR_2_PWR);

           //heater 1 actual value                   
           "AV".ACT_HTR_1_PWR           :=  #PM_INJET_HTR.htr_1_act_pwr; 
           "AV".ACT_HTR_1_CUR           :=  #PM_INJET_HTR.htr_1_act_cur; 
           "AV".ACT_HTR_1_VLT           :=  #PM_INJET_HTR.htr_1_act_vlt;
           "DIS".ACT_HTR1_ETH_VLT_PLUS  :=  #PM_INJET_HTR.htr_1_eth_vlt_plus;   // Erdschluss黚erwachung 
           "DIS".ACT_HTR1_ETH_VLT_MINUS :=  #PM_INJET_HTR.htr_1_eth_vlt_minus;  

           "FLT".HTR1_COMM_ERR       :=  #PM_INJET_HTR.htr_1_flt_comm;
           "FLT".HTR2_COMM_ERR       :=  #PM_INJET_HTR.htr_2_flt_comm;  
           "FLT".HTR1_RCT_TMP        :=  #PM_INJET_HTR.flt_htr1_rct_tmp; // temperature monitoring for heater 1 power supply filter reactor, limit by 85癈

           "FLT".HTR1_RCT_TMP        :=  #PM_INJET_HTR.flt_htr2_rct_tmp; // temperature monitoring for heater 2 power supply filter reactor, limit by 85癈

           "FLT".PWR_SPL_APF_ERR     :=  #PM_INJET_HTR.flt_pwr_spl_APF;
           "FLT".PWR_SPL_CTL_ERR     :=  #PM_INJET_HTR.htr_1_flt_ctrl OR #PM_INJET_HTR.htr_2_flt_ctrl;// 
           "FLT".HTR_1_ETH           :=  #PM_INJET_HTR.htr_1_flt_erd_plus OR #PM_INJET_HTR.htr_1_flt_erd_min;
           "FLT".HTR_2_ETH           :=  #PM_INJET_HTR.htr_2_flt_erd_plus OR #PM_INJET_HTR.htr_2_flt_erd_min;

           "AV".ACT_HTR_2_PWR           :=  #PM_INJET_HTR.htr_2_act_pwr; 
           "AV".ACT_HTR_2_CUR           :=  #PM_INJET_HTR.htr_2_act_cur; 
           "AV".ACT_HTR_2_VLT           :=  #PM_INJET_HTR.htr_2_act_vlt;
           "DIS".ACT_HTR2_ETH_VLT_PLUS  :=  #PM_INJET_HTR.htr_2_eth_vlt_plus;   // Erdschluss黚erwachung 
           "DIS".ACT_HTR2_ETH_VLT_MINUS :=  #PM_INJET_HTR.htr_2_eth_vlt_minus;  


           #flt_pwr_spl_panel_comm  := #PM_INJET_HTR.flt_pwr_spl_panel_comm;
           #htr_1_remote            := #PM_INJET_HTR.htr_1_remote;
           #comm_ok                 := #PM_INJET_HTR.comm_ok;
           #htr_pwr_spl_cool_wtr_flt:= #PM_INJET_HTR.htr_pwr_spl_cool_wtr_flt;
           #htr_pwr_spl_cool_wtr_wrn:= #PM_INJET_HTR.htr_pwr_spl_cool_wtr_wrn;


           #htr_1_flt_save          := #PM_INJET_HTR.htr_1_flt_save;
           #htr_1_flt_ac_pha        := #PM_INJET_HTR.htr_1_flt_ac_pha;
           #htr_1_flt_tmp           := #PM_INJET_HTR.htr_1_flt_tmp;
           #htr_1_flt_cur           := #PM_INJET_HTR.htr_1_flt_cur;
           #htr_1_flt_cool_wtr      := #PM_INJET_HTR.htr_1_flt_cool_wtr;
           #htr_1_flt_term          := #PM_INJET_HTR.htr_1_flt_term;
           #htr_1_mod1_flt_syn_kab := #PM_INJET_HTR.htr_1_mod1_flt_syn_kab;
           #htr_1_mod1_flt_sys_tmp := #PM_INJET_HTR.htr_1_mod1_flt_sys_tmp;
           #htr_1_mod1_flt_drv     := #PM_INJET_HTR.htr_1_mod1_flt_drv;
           #htr_1_mod1_flt_cur     := #PM_INJET_HTR.htr_1_mod1_flt_cur;
           #htr_1_mod1_flt_vlt     := #PM_INJET_HTR.htr_1_mod1_flt_vlt;
           #htr_1_mod1_flt_save    := #PM_INJET_HTR.htr_1_mod1_flt_save;
           #htr_1_mod1_flt_rect    := #PM_INJET_HTR.htr_1_mod1_flt_rect;
           #htr_1_mod1_flt_tmp     := #PM_INJET_HTR.htr_1_mod1_flt_tmp;


           #htr_1_mod2_flt_syn_kab := #PM_INJET_HTR.htr_1_mod2_flt_syn_kab;
           #htr_1_mod2_flt_sys_tmp := #PM_INJET_HTR.htr_1_mod2_flt_sys_tmp;
           #htr_1_mod2_flt_drv     := #PM_INJET_HTR.htr_1_mod2_flt_drv;
           #htr_1_mod2_flt_cur     := #PM_INJET_HTR.htr_1_mod2_flt_cur;
           #htr_1_mod2_flt_vlt     := #PM_INJET_HTR.htr_1_mod2_flt_vlt;
           #htr_1_mod2_flt_save    := #PM_INJET_HTR.htr_1_mod2_flt_save;
           #htr_1_mod2_flt_rect    := #PM_INJET_HTR.htr_1_mod2_flt_rect;
           #htr_1_mod2_flt_tmp     := #PM_INJET_HTR.htr_1_mod2_flt_tmp;


           #htr_1_mod3_flt_syn_kab := #PM_INJET_HTR.htr_1_mod3_flt_syn_kab;
           #htr_1_mod3_flt_sys_tmp := #PM_INJET_HTR.htr_1_mod3_flt_sys_tmp;
           #htr_1_mod3_flt_drv     := #PM_INJET_HTR.htr_1_mod3_flt_drv;
           #htr_1_mod3_flt_cur     := #PM_INJET_HTR.htr_1_mod3_flt_cur;
           #htr_1_mod3_flt_vlt     := #PM_INJET_HTR.htr_1_mod3_flt_vlt;
           #htr_1_mod3_flt_save    := #PM_INJET_HTR.htr_1_mod3_flt_save;
           #htr_1_mod3_flt_rect    := #PM_INJET_HTR.htr_1_mod3_flt_rect;
           #htr_1_mod3_flt_tmp     := #PM_INJET_HTR.htr_1_mod3_flt_tmp;

           #htr_1_mod4_flt_syn_kab := #PM_INJET_HTR.htr_1_mod4_flt_syn_kab;
           #htr_1_mod4_flt_sys_tmp := #PM_INJET_HTR.htr_1_mod4_flt_sys_tmp;
           #htr_1_mod4_flt_drv     := #PM_INJET_HTR.htr_1_mod4_flt_drv;
           #htr_1_mod4_flt_cur     := #PM_INJET_HTR.htr_1_mod4_flt_cur;
           #htr_1_mod4_flt_vlt     := #PM_INJET_HTR.htr_1_mod4_flt_vlt;
           #htr_1_mod4_flt_save    := #PM_INJET_HTR.htr_1_mod4_flt_save;
           #htr_1_mod4_flt_rect    := #PM_INJET_HTR.htr_1_mod4_flt_rect;
           #htr_1_mod4_flt_tmp     := #PM_INJET_HTR.htr_1_mod4_flt_tmp;  

           #htr_2_remote           := #PM_INJET_HTR.htr_2_remote;
           #htr_2_flt_save         := #PM_INJET_HTR.htr_2_flt_save;
           #htr_2_flt_ac_pha       := #PM_INJET_HTR.htr_2_flt_ac_pha;
           #htr_2_flt_tmp          := #PM_INJET_HTR.htr_2_flt_tmp;
           #htr_2_flt_cur          := #PM_INJET_HTR.htr_2_flt_cur;
           #htr_2_flt_cool_wtr     := #PM_INJET_HTR.htr_2_flt_cool_wtr;
           #htr_2_flt_term         := #PM_INJET_HTR.htr_2_flt_term;
           #htr_2_mod1_flt_syn_kab := #PM_INJET_HTR.htr_2_mod1_flt_syn_kab;
           #htr_2_mod1_flt_sys_tmp := #PM_INJET_HTR.htr_2_mod1_flt_sys_tmp;
           #htr_2_mod1_flt_drv     := #PM_INJET_HTR.htr_2_mod1_flt_drv;
           #htr_2_mod1_flt_cur     := #PM_INJET_HTR.htr_2_mod1_flt_cur;
           #htr_2_mod1_flt_vlt     := #PM_INJET_HTR.htr_2_mod1_flt_vlt;
           #htr_2_mod1_flt_save    := #PM_INJET_HTR.htr_2_mod1_flt_save;
           #htr_2_mod1_flt_rect    := #PM_INJET_HTR.htr_2_mod1_flt_rect;
           #htr_2_mod1_flt_tmp     := #PM_INJET_HTR.htr_2_mod1_flt_tmp;

           #htr_2_mod2_flt_syn_kab := #PM_INJET_HTR.htr_2_mod2_flt_syn_kab;
           #htr_2_mod2_flt_sys_tmp := #PM_INJET_HTR.htr_2_mod2_flt_sys_tmp;
           #htr_2_mod2_flt_drv     := #PM_INJET_HTR.htr_2_mod2_flt_drv;
           #htr_2_mod2_flt_cur     := #PM_INJET_HTR.htr_2_mod2_flt_cur;
           #htr_2_mod2_flt_vlt     := #PM_INJET_HTR.htr_2_mod2_flt_vlt;
           #htr_2_mod2_flt_save    := #PM_INJET_HTR.htr_2_mod2_flt_save;
           #htr_2_mod2_flt_rect    := #PM_INJET_HTR.htr_2_mod2_flt_rect;
           #htr_2_mod2_flt_tmp     := #PM_INJET_HTR.htr_2_mod2_flt_tmp;

           #htr_2_mod3_flt_syn_kab := #PM_INJET_HTR.htr_2_mod3_flt_syn_kab;
           #htr_2_mod3_flt_sys_tmp := #PM_INJET_HTR.htr_2_mod3_flt_sys_tmp;
           #htr_2_mod3_flt_drv     := #PM_INJET_HTR.htr_2_mod3_flt_drv;
           #htr_2_mod3_flt_cur     := #PM_INJET_HTR.htr_2_mod3_flt_cur;
           #htr_2_mod3_flt_vlt     := #PM_INJET_HTR.htr_2_mod3_flt_vlt;
           #htr_2_mod3_flt_save    := #PM_INJET_HTR.htr_2_mod3_flt_save;
           #htr_2_mod3_flt_rect    := #PM_INJET_HTR.htr_2_mod3_flt_rect;
           #htr_2_mod3_flt_tmp     := #PM_INJET_HTR.htr_2_mod3_flt_tmp;

       END_IF;

       //set display values
       //------------------                  
       IF #htr_1_enb  THEN
           "DIS".ACT_HTR_1_PWR   :=  "AV".ACT_HTR_1_PWR;
           "DIS".ACT_HTR_1_CUR   :=  "AV".ACT_HTR_1_CUR;
           "DIS".ACT_HTR_1_VLT   :=  "AV".ACT_HTR_1_VLT;
           "DIS".ACT_HTR_1_ETH_FLT_VAL := (("P_BM_ETH_FLT_MON_IIST1":P-"P_BM_ETH_FLT_MON_UIST1":P)/4095.0) *100.0;  // Scaled on 100% >>only Plating power supply
       ELSE
           "DIS".ACT_HTR_1_PWR   :=  0.0;
           "DIS".ACT_HTR_1_CUR   :=  0.0;
           "DIS".ACT_HTR_1_VLT   :=  0.0;
           "DIS".ACT_HTR_1_ETH_FLT_VAL := 0.0;
       END_IF;


       //set display values
       //------------------                  
       IF #htr_2_enb  THEN
           "DIS".ACT_HTR_2_PWR   :=  "AV".ACT_HTR_2_PWR;
           "DIS".ACT_HTR_2_CUR   :=  "AV".ACT_HTR_2_CUR;
           "DIS".ACT_HTR_2_VLT   :=  "AV".ACT_HTR_2_VLT;
           "DIS".ACT_HTR_2_ETH_FLT_VAL := (("P_BM_ETH_FLT_MON_IIST2":P-"P_BM_ETH_FLT_MON_UIST2":P)/4095.0) *100.0;  // Scaled on 100% >>only Plating power supply 
       ELSE
           "DIS".ACT_HTR_2_PWR   :=  0.0;
           "DIS".ACT_HTR_2_CUR   :=  0.0;
           "DIS".ACT_HTR_2_VLT   :=  0.0;
           "DIS".ACT_HTR_2_ETH_FLT_VAL :=  0.0;
       END_IF;
END_FUNCTION_BLOCK

FUNCTION_BLOCK "BM_HTR_RES_CALC"   // FB70, SCL
{ S7_Optimized_Access := 'FALSE' }
VERSION : 0.0
// --------------------------------------------------------------------------------------
//     program     :    BM_RES_CALC
//     description :    calculate heater resistance 
//     name        :    G. Eibelsh鋟ser
//     date        :    11.10.2005
// 
//     revision    :
//     name        :
//     date        :    
//                     
//                     (c)PVATepla AG
//     --------------------------------------------------------------------------------------
   VAR_INPUT
      pwr_set : Real;
      act_pwr : Real;
      act_cur : Real;
      act_vlt : Real;
   END_VAR
   VAR_IN_OUT
      res_act : Real;
      res_change : Real;
   END_VAR
   VAR
      i : Int;
      res_old : Real;
      pwr_set_old : Real;
   END_VAR
   VAR CONSTANT
      pwr_max_dev : Real := 2.0;
   END_VAR
BEGIN


       IF ABS(#pwr_set - #pwr_set_old) > #pwr_max_dev THEN
           #i:= 0;
       END_IF;
       IF (#act_pwr > #pwr_max_dev) THEN
           IF (#i > 5) THEN      
             //res_act     := 1000.0 * act_pwr / act_cur**2;       //r = p / i^2 (range is OHM)
               #res_act     := #act_vlt / #act_cur;                   //r = U / i
               #res_change  := #res_act - #res_old;               //r change
           ELSE 
               #res_change := 0.0;
               #i := #i+ 1;
           END_IF;    
       ELSE
           #res_act     := 0.0;
           #res_change  := 0.0;
       END_IF;

       #pwr_set_old := #pwr_set;                                        //save previous values
       #res_old     := #res_act;
END_FUNCTION_BLOCK

FUNCTION_BLOCK "BM_CALL_RES_CALC"   // FB71, SCL
{ S7_Optimized_Access := 'FALSE' }
VERSION : 0.0
// --------------------------------------------------------------------------------
//     program     :    BM_CALL_RES_CALC (1000ms interrupt)
//     description :    call all modules for power supply resistance calculation 
//     name        :    L.Vogel
//     date        :    25.06.2018
// 
//     revision    :   GCL injet Power Supply
//     name        :   John Wang
//     date        :   18.08.2020
//     
//                     (c)PVA CGS GmbH
//     --------------------------------------------------------------------------------
   VAR
      BM_RES_HTR_1 : "BM_HTR_RES_CALC";
      BM_RES_HTR_2 : "BM_HTR_RES_CALC";
   END_VAR
BEGIN

       //call resistance calculation of heater 1
       //---------------------------------------
       #BM_RES_HTR_1(   res_act     := "AV".ACT_HTR_1_RES,
                       res_change  := "AV".ACT_HTR_1_RES_CNG,
                       pwr_set     := "CTL".SET_HTR_1_PWR,
                       act_pwr     := "DIS".ACT_HTR_1_PWR,
                       act_cur     := "AV".ACT_HTR_1_CUR,
                       act_vlt     := "AV".ACT_HTR_1_VLT); 

       //set display value
       //-----------------                

       IF  "CNF".CONF_PWR_SPL_TYPE = 1 THEN     

           "DIS".ACT_HTR_1_RES   :=   "AV".ACT_HTR_1_RES * 1000.0;     //range of display value is mOHM    

       END_IF;

       IF  "CNF".CONF_PWR_SPL_TYPE = 2 THEN  

           "DIS".ACT_HTR_1_RES   := "P_BM_PWR_SPL_1_ACT_RESIS":P * 1000.0;   // Injet act. resistance [mOHM]

       END_IF; 


       //call resistance calculation of heater 2
       //---------------------------------------
       #BM_RES_HTR_2(   res_act     := "AV".ACT_HTR_2_RES,
                       res_change  := "AV".ACT_HTR_2_RES_CNG,
                       pwr_set     := "CTL".SET_HTR_2_PWR,
                       act_pwr     := "DIS".ACT_HTR_2_PWR,
                       act_cur     := "AV".ACT_HTR_2_CUR,
                       act_vlt     := "AV".ACT_HTR_2_VLT); 

        //set display value
        //-----------------                

       IF  "CNF".CONF_PWR_SPL_TYPE = 1 THEN     

           "DIS".ACT_HTR_2_RES   :=   "AV".ACT_HTR_2_RES * 1000.0;           //range of display value is mOHM     

       END_IF;

       IF  "CNF".CONF_PWR_SPL_TYPE = 2 THEN  

           "DIS".ACT_HTR_2_RES   := "P_BM_PWR_SPL_2_ACT_RESIS":P * 1000.0;  // Injet act. resistance [mOHM]

       END_IF;
END_FUNCTION_BLOCK

FUNCTION_BLOCK "BM_ROT_DRV_DIR"   // FB72, SCL
{ S7_Optimized_Access := 'FALSE' }
VERSION : 0.0
// --------------------------------------------------------------------------------
//     program     :    BM_ROT_DRV_DIR
//     description :    rotation drive direction in automatic mode 
//     name        :    G. Eibelsh鋟ser
//     date        :    06.06.2000
//     
//                         ROT_DIR = 0  ,  XT = ccw, CR = CW
//                         ROT_DIR = 1  ,  XT =  cw, CR = CCW
// 
//     revision    :
//     name        :
//     date        :    
//                     (c)CGS
//     --------------------------------------------------------------------------------
   VAR
      ROT_DIR : Bool;
   END_VAR
BEGIN


       IF "LT".XT_ROT_OFF AND "LT".CR_ROT_OFF  THEN
           #ROT_DIR :=  "PAR_MAIN".MCONST_ROT_DIR = 1.0;
       ELSE      
           IF #ROT_DIR = TRUE THEN
               "PAR_MAIN".MCONST_ROT_DIR := 1.0;
           ELSE    
               "PAR_MAIN".MCONST_ROT_DIR := 0.0;
           END_IF;
       END_IF;
END_FUNCTION_BLOCK

FUNCTION_BLOCK "BM_MAG"   // FB75, SCL
{ S7_Optimized_Access := 'FALSE' }
VERSION : 0.0
// --------------------------------------------------------------------------------
//     program     :    BM_MAG
//     description :    basic functions magnet
//                      
//  
//     name        :    L.Vogel
//     date        :    18.05.2011
// 
//     revision    :    CGS1218 mit Simitomo magnet
//     name        :    John Wang
//     date        :    15.03.2019 
//      
//                     (c)PVATEPLA
//     --------------------------------------------------------------------------------
   VAR
      MAG_CTRL_OUT : Word;
      MAG_OUT AT MAG_CTRL_OUT : Struct
         B00_EMO : Bool;   // ON : Emergency stop
         B01_FLT_ACK : Bool;   // Reset
         B02_SET_CUR : Bool;   // Permit current set ( level command )
         B03_Spare : Bool;
         B04_CUR_OFF : Bool;   // set current to 0.0A
         B05_Spare : Bool;
         B06_Spare : Bool;
         B07_Spare : Bool;
         B10_Spare : Bool;
         B11_Spare : Bool;
         B12_Spare : Bool;
         B13_Spare : Bool;
         B14_Spare : Bool;
         B15_Spare : Bool;
         B16_Spare : Bool;
         B17_Spare : Bool;
      END_STRUCT;
      MAG_SET_CUR : Int;
      MAG_STAT_IN : Word;
      MAG_STAT AT MAG_STAT_IN : Struct
         B00_PWR_FLT : Bool;   // Power failure (necessary to reset)
         B01_EMG_DEM : Bool;   // Emergency demagnetize (necessary to reset)
         B02_RDY : Bool;   // Remote, ON, Coil normal temp.normal and Shield temp.normal
         B03_EXC : Bool;   // Excitation
         B04_REMOTE : Bool;   // ON : Remote operation OFF: Local operation
         B05_PWR_SLY_FLT : Bool;   // Power supply fault (necessary to reset)
         B06_Quench : Bool;   // Quench (necessary to reset)
         B07_Spare : Bool;
         B10_Spare : Bool;
         B11_Spare : Bool;
         B12_Spare : Bool;
         B13_Spare : Bool;
         B14_Spare : Bool;
         B15_Spare : Bool;
         B16_Spare : Bool;
         B17_Spare : Bool;
      END_STRUCT;
      MAG_STAT2_IN : Word;
      MAG_STAT2 AT MAG_STAT2_IN : Struct
         B10_COMP_A1_ON : Bool;   // compressor unit 1 drive
         B11_COMP_A2_ON : Bool;   // compressor unit 2 drive
         B12_COMP_B1_ON : Bool;   // compressor unit 3 drive
         B13_COMP_B2_ON : Bool;   // compressor unit 4 drive
         B14_COMP_A1_PRS : Bool;   // compressor unit 1 Pressure fault
         B15_COMP_A2_PRS : Bool;   // compressor unit 2 Pressure fault
         B16_COMP_B1_PRS : Bool;   // compressor unit 3 Pressure fault
         B17_COMP_B2_PRS : Bool;   // compressor unit 4 Pressure fault
         B20_COMP_A1_TMP : Bool;   // compressor unit 1 temperature fault
         B21_COMP_A2_TMP : Bool;   // compressor unit 2 temperature fault
         B22_COMP_B1_TMP : Bool;   // compressor unit 3 temperature fault
         B23_COMP_B2_TMP : Bool;   // compressor unit 4 temperature fault
         B24_Spare : Bool;
         B25_Spare : Bool;
         B26_Spare : Bool;
         B27_Spare : Bool;
      END_STRUCT;
      MAG_STAT3_IN : Word;
      MAG_STAT3 AT MAG_STAT3_IN : Struct
         B30_FLT_TMP_COIL_1 : Bool;   // magnet coil 1 temperature fault
         B31_FLT_TMP_COIL_2 : Bool;   // magnet coil 2 temperature fault (necessary to reset)
         B32_FLT_TMP_SHLD_1 : Bool;   // radiation shield 1 temperature fault
         B33_FLT_TMP_SHLD_2 : Bool;   // radiation shield 2 temperature fault (necessary to reset)
         B34_Spare : Bool;
         B35_Spare : Bool;
         B36_Spare : Bool;
         B37_Spare : Bool;
         B40_Spare : Bool;
         B41_Spare : Bool;
         B42_Spare : Bool;
         B43_Spare : Bool;
         B44_Spare : Bool;
         B45_Spare : Bool;
         B46_Spare : Bool;
         B47_Spare : Bool;
      END_STRUCT;
      MAG_ACT_CUR : Int;
      MAG_ACT_VLT : Int;
      MAG_ACT_TMP_COIL_A1 : Int;
      MAG_ACT_TMP_COIL_A2 : Int;
      MAG_ACT_TMP_COIL_B1 : Int;
      MAG_ACT_TMP_COIL_B2 : Int;
      MAG_ACT_TMP_SHLD : Int;
      mag_stby_itl_ok : Bool;
      MAG_STBY_ON : Bool;
      MAG_STBY_OFF_DLY : Bool;
      mag_itl_ok : Bool;
      MAG_ON : Bool;
      MAG_OFF_DLY : Bool;
      flt_magnet : Bool;
      TimeStbyOff : Int;
      TimeMagOff : Int;
      TMP_VAL : Int;
      set_cur1 : Real;
      set_cur2 : Real;
      ratio_cur2 : Real;
      "b" : Real;
   END_VAR
BEGIN

       //read values from magnet
       //-------------------------------------
       #MAG_STAT_IN  := BYTE_TO_WORD("P_BM_MAG_STAT":P);
       #MAG_STAT2_IN := "P_BM_MAG_STAT2":P;
       #MAG_STAT3_IN := BYTE_TO_WORD("P_BM_MAG_STAT3":P);
       #MAG_ACT_CUR  := WORD_TO_INT("P_BM_MAG_ACT_CUR":P);
       #MAG_ACT_VLT  := WORD_TO_INT("P_BM_MAG_ACT_VLT":P);
       #MAG_ACT_TMP_COIL_A1 := WORD_TO_INT("P_BM_MAG_ACT_TMP_COIL_A1":P);
       #MAG_ACT_TMP_COIL_A2 := WORD_TO_INT("P_BM_MAG_ACT_TMP_COIL_A2":P);
       #MAG_ACT_TMP_COIL_B1 := WORD_TO_INT("P_BM_MAG_ACT_TMP_COIL_B1":P);
       #MAG_ACT_TMP_COIL_B2 := WORD_TO_INT("P_BM_MAG_ACT_TMP_COIL_B2":P);
       #MAG_ACT_TMP_SHLD    := WORD_TO_INT("P_BM_MAG_ACT_TMP_SHLD":P);

       //set fault message in process and bake out state
       //-----------------------------------------------
       IF (("STA".ACT_STATE = "APC".STATE_RUN) OR ("STA".ACT_STATE = "APC".STATE_BAKE_OUT)) THEN
           "FLT".MAG_LFT_NOT_IN_POS := "DC".MAG_ON AND NOT "PDI".LS_MAG_LFT_UP;    
       //set fault message in manual mode when key is touched
       //----------------------------------------------------
       ELSIF "LT".MOD_MANUAL THEN
           "FLT".MAG_LFT_NOT_IN_POS := "KYD".MAG_ON AND NOT "PDI".LS_MAG_LFT_UP;    
       //reset
       //-----
       ELSE
           "FLT".MAG_LFT_NOT_IN_POS := FALSE;
       END_IF;

       //build set point
       //---------------
       IF "KYA".SET_MAG_1_CUR > "CNF".MAG_1_CUR_RANGE THEN   // Max 170.0A 
           "KYA".SET_MAG_1_CUR := "CNF".MAG_1_CUR_RANGE;
       END_IF;
       IF "AC".SET_MAG_1_CUR > "CNF".MAG_1_CUR_RANGE THEN
           "AC".SET_MAG_1_CUR := "CNF".MAG_1_CUR_RANGE;
       END_IF;

       #set_cur1    := "CM_INSELECT"(auto  := "APC".AUTOMATIC AND NOT "SY".CTL_MAG_1_SMI,            
                                 track := true,
                                 ac    := "AC".SET_MAG_1_CUR,
                                 kya   := "KYA".SET_MAG_1_CUR);


       #ratio_cur2 := "CM_INSELECT"(auto  := "APC".AUTOMATIC AND NOT "SY".CTL_MAG_1_SMI,            
                                 track := true,
                                 ac    := "AC".SET_MAG_RATIO_CUR,
                                 kya   := "KYA".SET_MAG_RATIO_CUR);

       IF "KYA".SET_MAG_RATIO_CUR < 0.5 THEN
           "KYA".SET_MAG_RATIO_CUR := 1.0;
       ELSE
           IF ("KYA".SET_MAG_RATIO_CUR> 1.5) OR (("KYA".SET_MAG_RATIO_CUR * "KYA".SET_MAG_1_CUR)>"CNF".MAG_1_CUR_RANGE) THEN
               "KYA".SET_MAG_RATIO_CUR := 1.0;
           END_IF;
       END_IF;

       //build set point coil2
       #set_cur2 := #set_cur1 * #ratio_cur2;
       IF #set_cur2> "CNF".MAG_1_CUR_RANGE THEN
           #set_cur2 := "CNF".MAG_1_CUR_RANGE;
       END_IF;

       //magnet interlock bit
       //--------------------
       #mag_itl_ok := "PDI".EMO AND "PDI".LS_MAG_LFT_UP;

       //magnet on/off
       //-------------                    
       "CM_ITL_IO"(ADR := 61,
              KYD_ON := "KYD".MAG_ON,
              KYD_OFF:= "KYD".MAG_OFF,
              AUTO := "APC".AUTOMATIC,
              DC_ON:= "DC".MAG_ON,
              CON1 := #mag_itl_ok, 
              CON2 := "SysLog1", //MAG_STAT.B04_REMOTE OR MAG_ON, 
              CON3 := NOT #flt_magnet,
              CON4 := "SysLog1",
              CON5 := "SysLog1",
              CON6 := "SysLog1",
              CON7 := "SysLog1",
              CON8 := "SysLog1",
              ITL_OUT:= "STA_ITL_CAUSE",
              LT_OUT := #MAG_ON);

       "LT".MAG_ON      := #MAG_ON;

       #MAG_OFF_DLY := "SysOffdelay"( DIN := NOT #MAG_ON AND ("DIS".ACT_MAG_1_CUR< 1.0),
                                   SetTime := 3,                           // setp. time
                                   ActTime := #TimeMagOff,                   // act. time
                                   Tick    := "SysTick1s"    );              // timebase (1s)

       #MAG_OUT.B04_CUR_OFF := #MAG_OFF_DLY;
       #MAG_OUT.B02_SET_CUR := #MAG_ON;

       //reset power setpoint if heater enable is gone
       //---------------------------------------------
       #MAG_OUT.B01_FLT_ACK := "KYD".MAG_TRIP_RES;
       #MAG_OUT.B00_EMO     := NOT "PDI".EMO;


       //write set points
       //----------------
      IF #MAG_OUT.B02_SET_CUR THEN
           #MAG_SET_CUR   := REAL_TO_INT(#set_cur1*10.0);
       ELSE
          #MAG_SET_CUR   := 0;
          "KYA".SET_MAG_1_CUR   := 0.0; 
       END_IF;


       //check fault conditions 
       //----------------------
         //check fault conditions 
       //----------------------
       "FLT".MAG_PWR_SPL   :=  #MAG_STAT.B05_PWR_SLY_FLT;        //  Power failure  (necessary to reset)
       "FLT".MAG_QUENCH    :=  #MAG_STAT.B06_Quench;             //Quench
       "FLT".MAG_EMG_OFF   :=  #MAG_STAT.B01_EMG_DEM;            //Notabschaltung
       "FLT".MAG_MAIN_LINE :=  #MAG_STAT.B00_PWR_FLT;             //Stromausfall
       "FLT".MAG_TMP       :=  #MAG_STAT3.B30_FLT_TMP_COIL_1 OR #MAG_STAT3.B31_FLT_TMP_COIL_2 OR #MAG_STAT3.B32_FLT_TMP_SHLD_1 OR #MAG_STAT3.B33_FLT_TMP_SHLD_2;             //Temperatur
       "FLT".MAG_CUR_FEED  :=  FALSE;
       "FLT".MAG_VAC       :=  #MAG_STAT2.B14_COMP_A1_PRS OR #MAG_STAT2.B15_COMP_A2_PRS OR #MAG_STAT2.B16_COMP_B1_PRS OR #MAG_STAT2.B17_COMP_B2_PRS;              //Vakuum
       "FLT".MAG_HE_COMPR  :=  #MAG_STAT2.B20_COMP_A1_TMP OR #MAG_STAT2.B21_COMP_A2_TMP OR #MAG_STAT2.B22_COMP_B1_TMP OR #MAG_STAT2.B23_COMP_B2_TMP;        //HE-Kompressoren
       "FLT".WRN_MAG       :=  FALSE;               

       #flt_magnet        := "FLT".MAG_PWR_SPL OR "FLT".MAG_QUENCH OR "FLT".MAG_EMG_OFF OR "FLT".MAG_MAIN_LINE OR 
                            "FLT".MAG_TMP OR "FLT".MAG_CUR_FEED OR "FLT".MAG_VAC OR "FLT".MAG_HE_COMPR;

       IF "AV".SET_MAG_1_CUR > "CNF".MAG_1_CUR_RANGE THEN
           "AV".SET_MAG_1_CUR := "CNF".MAG_1_CUR_RANGE;
           "FLT".PAR_FLT_MAG_1_CUR :=  TRUE;
       ELSE
           "FLT".PAR_FLT_MAG_1_CUR :=  FALSE;
       END_IF;      

       //write display value
       //------------------------
       IF NOT #MAG_OFF_DLY THEN 
           "DIS".SET_MAG_1_CUR   := #set_cur1;
           "DIS".ACT_MAG_1_CUR   := INT_TO_REAL(#MAG_ACT_CUR)/10.0;   
           "DIS".ACT_MAG_1_VLT   := INT_TO_REAL(#MAG_ACT_VLT)/10.0;   
       ELSE   
           "DIS".ACT_MAG_1_CUR   := 0.0;
           "DIS".ACT_MAG_1_VLT   := 0.0;
       END_IF;    
      (* Logik Magneten zum Status 
         ----------------------------------------
       00: s_OFF    Magnet aus, K黨lung aus
       10: s_PRECON    Magnet aus, K黨lung aktiv
       20: s_STANDBY    Magnet aus, K黨lung abgeschlossen
       30: s_OPERATION    Magnet ein, keine Fehler
       40: s_QUENCH    Magnetfeldverlust in <1s
       50: s_WARNING    Magnet ein, Warnung aktiv
       60: s_ERROR    Magnet wird automatisch 黚er Netzteil entladen (30MIN, aktive Entladung bei Temperatur, HTS oder Vakuumfehlern)
       70: s_DISCHARGE    Magnet wird passiv entladen (30MIN, passive Entladung bei Stromausfall oder Netzteilfehler)
       80: s_EMERGENCY    Magnet wird gequencht (Entladung in ca. 1s)
       90: s_PRE_WARNING    Magnet aus, Warnung von K黨lung oder Vakuum
      100: s_PRE_ERROR    Magnet aus, Fehler von K黨lung oder Vakuum
      --------------------------------------------
      *)

       IF "FLT".MAG_PWR_SPL OR "FLT".MAG_MAIN_LINE THEN      
           "DIS".ACT_MAG_STATE  := 60.0;
       ELSIF "FLT".MAG_QUENCH THEN
           "DIS".ACT_MAG_STATE  := 40.0;
       ELSIF "FLT".MAG_EMG_OFF THEN
           "DIS".ACT_MAG_STATE  := 80.0;
       ELSIF "FLT".MAG_VAC  OR  "FLT".MAG_HE_COMPR THEN
           "DIS".ACT_MAG_STATE  := 90.0;
       ELSIF "LT".MAG_ON THEN
           "DIS".ACT_MAG_STATE  := 30.0;
       ELSIF #MAG_STAT.B04_REMOTE AND  #MAG_STAT.B02_RDY THEN
           "DIS".ACT_MAG_STATE  := 20.0;
       ELSIF #MAG_STAT.B04_REMOTE THEN
           "DIS".ACT_MAG_STATE  := 10.0;
       ELSE
           "DIS".ACT_MAG_STATE  := 0.0;
       END_IF;

       //Write the hight value in the display value   
       #TMP_VAL  := #MAG_ACT_TMP_COIL_A1;
       IF #TMP_VAL < #MAG_ACT_TMP_COIL_A2 THEN 
          #TMP_VAL := #MAG_ACT_TMP_COIL_A2;
       END_IF;   
       IF #TMP_VAL < #MAG_ACT_TMP_COIL_B1 THEN
          #TMP_VAL := #MAG_ACT_TMP_COIL_B1;
       END_IF;   
       IF #TMP_VAL < #MAG_ACT_TMP_COIL_B2 THEN 
          #TMP_VAL := #MAG_ACT_TMP_COIL_B2;
       END_IF;

       IF NOT "SY".SIM_ON THEN 
          "DIS".ACT_MAG_1_TMP  := INT_TO_REAL(#TMP_VAL);
       END_IF;          
       IF "DIS".ACT_MAG_1_CUR<15.0 THEN
           #b := 136.0 *"DIS".ACT_MAG_1_CUR/15.0;
       ELSE
           #b := 136.0;    
       END_IF;          
       "DIS".ACT_MAG_FLD    := ("DIS".ACT_MAG_1_CUR * 23.2) + #b;        // y=mx+b => (Feld[Gs] = Current[A] * 23.2 + 136); Acordding messure protokol Sumitomo
       "DIS".ACT_MAG_POS  := 850.0*INT_TO_REAL("STA".MAG_LFT_POS)/100.0; // Max Lift Pos * calculate position in %

      //write values to interface
      //-------------------------
      "P_BM_MAG_CTRL":P    := WORD_TO_BYTE(SHR(IN :=#MAG_CTRL_OUT,N :=8));
      "P_BM_MAG_SET_CUR":P := INT_TO_WORD(#MAG_SET_CUR);
END_FUNCTION_BLOCK

FUNCTION_BLOCK "BM_SEED_TMP_CTL"   // FB86, SCL
{ S7_Optimized_Access := 'FALSE' }
VERSION : 0.0
// ---------------------------------------------------------------------------------
//     program     :    BM_SEED_TMP_CTL
//     description :    monitoring of seed temp to stop xt_lft when seed is hot (manual mode)
//     
//     name        :    M.Lech
//     date        :    19.02.2003
//     
// 
//     revision    :
//     name        :
//     date        :    
//                     (c)CGS
//     ---------------------------------------------------------------------------------
   VAR
      seed_cool_dn_act_tme : Int;   // actual time for cool down wait time
      seed_cool_dn_set_tme : Int;   // setpoint for cool down wait time
      seed_hot : Bool;   // detection seed hot
      seed_cool_dn_dly : Bool;
      XT_LFT_FST_OFF : Bool;   // flag to switch xt speed from fast to normal
      XT_LFT_OFF : Bool;   // flag to switch xt lft off
   END_VAR
BEGIN

       #seed_cool_dn_set_tme := 30 * 60;    // setpoint cool down wait time [s]

       IF ("AV".ACT_XT_POS > "CNF".SEED_TMP_CTL_POS_LIM) AND              // xt below limit? 
           ("AV".ACT_HTR_1_TMP > "CNF".HTR_1_TMP_RANGE_LOW + 10.0)  THEN   // heater temp. higher than min. value?
           #seed_hot := TRUE;
       ELSE
           #seed_hot := FALSE;
       END_IF;


       // start timer when seed is cooling down (heater temp. below limit or xt position above limit)
       // -------------------------------------------------------------------------------------------
       #seed_cool_dn_dly := "SysOffdelay"(SetTime := #seed_cool_dn_set_tme,        // IN: INT
                                       Tick    := "SysTick1s",                   // IN: BOOL
                                       DIN     := #seed_hot,                    // IN: BOOL
                                       ActTime := #seed_cool_dn_act_tme);       // INOUT: INT




       #XT_LFT_FST_OFF := ("AV".ACT_XT_POS <= ("CNF".SEED_TMP_CTL_HI_POS + "CNF".xt_lft_rmp))         // switch FAST mode off x mm before stop position
                           AND #seed_cool_dn_dly;                                               // do not switch off if dly time for cooling down is over

       #XT_LFT_OFF := #seed_cool_dn_dly                                                          // do not switch off if dly time for cooling down is over        
                       AND ("AV".ACT_XT_POS <= "CNF".SEED_TMP_CTL_HI_POS);                        // switch xt lift off if stop position is reached


       IF #XT_LFT_OFF THEN
          "FLT".SEED_TMP := TRUE;
       ELSE
          "FLT".SEED_TMP := FALSE;
       END_IF;
END_FUNCTION_BLOCK

FUNCTION_BLOCK "BM_SI_FIL_REG"   // FB88, SCL
{ S7_Optimized_Access := 'FALSE' }
VERSION : 0.0
// -----------------------------------------------------------------------------------
//     program:         BM_SI_FIL_REG
//     description :    Silicon filter regeneration
//     name:            G. Eibelsh鋟ser
//     date        :    10.08.2011
// 
//     revision    :   CGS 1218 
//     name        :   J. Wang
//     Date        :   09.12.2019
//     
//    
//     
//                     (c)PVA TePla AG
// -----------------------------------------------------------------------------------
   VAR
      req_fil_cln : Bool;
      run_fil_cln : Bool;
      fill_up_sto_tank : Bool;
      "step" : Int;
      i : Int;
      count : Int;
      act_state_prev : Int;
   END_VAR
BEGIN


       //abort filter cleaning sequence
       //--------------------------------
       IF ("KYD".SI_FIL_FSH_SEQ_OFF OR ("APC".STATUS <> "APC".IDLE) OR "DV".FIL_CLN_REQ_IN_PRC) THEN
           #req_fil_cln :=  false;

       //request filter cleaning sequence
       //--------------------------------
       ELSIF ("KYD".SI_FIL_FSH_SEQ_ON OR "DV".FIL_FSH_REQ_AFTER_SD) THEN
           #req_fil_cln :=  true;
       END_IF;

       //set light variable filter flushing sequence
       //-------------------------------------------    
       IF #req_fil_cln THEN 
           #run_fil_cln             :=  true;       //enable filter flushing
           "FLT".SI_FIL_REG_ENB      :=  FALSE;      //reset alarm message when Si filter regeneration sequence is requested
           "DV".FIL_FSH_REQ_AFTER_SD :=  FALSE;      //reset flag filter regeneration after shut down 
       END_IF;

       //fill up gas storage tank
       //------------------------
       IF #fill_up_sto_tank THEN
           IF ("DIS".ACT_PRS_AR_VSL < "CNF".MAX_PRS_AR_VSL) THEN
               //open valve V25
               //--------------
               "DV".V25_OP   :=  TRUE;
           ELSE
               //close valve V25
               //--------------
               "DV".V25_OP           :=  FALSE;
               #fill_up_sto_tank    :=  false;  //fill up finished
           END_IF;
       END_IF;

       //do filter flushing sequence
       //---------------------------
       IF #run_fil_cln  THEN 
           IF NOT #req_fil_cln  AND (#step < 110) THEN       //abort cleaning sequence
               #step    :=  110;
               #i       :=   0;
           END_IF;

           //sequence steps
           //--------------
           CASE #step OF 

               0 : //initialisation step
                   //-------------------
                   "DC".V2_1_OP      :=  FALSE;      //close main vacuum valve to furnace
                   "DC".V3_OP        :=  FALSE;
                   "DC".V3_2_OP      :=  FALSE;
                   "DC".V4_OP        :=  FALSE;
                   "DC".V5_OP        :=  FALSE;
                   "DC".V6_OP        :=  FALSE;
                   "DC".V11_OP       :=  FALSE;
                   "DC".V19_OP       :=  FALSE;      //close dust outlet valve filter
                   "DC".V20_OP       :=  FALSE;
                   "DC".V21_OP       :=  FALSE;
                   "DC".V22_OP       :=  FALSE;      //close Ar inlet valve filter
                   "DC".V24_OP       :=  FALSE;
                   "DC".P1_ON        :=  TRUE;       //run vacuum pump
                   "DC".P3_ON        :=  FALSE;
                   "LT".SI_FIL_FSH_SEQ_ON    :=  TRUE;       //set illumination of button
                   #fill_up_sto_tank        :=  true;       //request fill up of storage tank
                   "AC".SET_GAS_1_FLW        :=  0.0;
                   "AC".SET_GAS_2_FLW        :=  0.0;

                   #count                   :=  0;
                   #i                       :=  0;

                   IF "BM_VAC_DB".P1_IS_ON THEN
                       "AC".SET_CTL_VALVE_POS    := "CTL".SET_CTL_VALVE_POS; 
                   ELSE
                       "AC".SET_CTL_VALVE_POS    := 0.0;
                   END_IF;

                   #step            :=  #step + 10;

               10: //set global aux flag regeneration sequence is active
                   //---------------------------------------------------
                   "DV".SI_FIL_FSH_SEQ_ON    :=  TRUE;                   //close request to valve V2.1

                   IF NOT "PDO".V2_1 THEN 
                       "AC".SET_CTL_VALVE_POS    :=  100.0;      //open pressure control valve

                       //pump down filter (120sec  after V1 completly open)
                       //--------------------------------------------------                    
                       IF ("DIS".ACT_CTL_VALVE_POS >= 98.0) THEN  
                           //count wait time
                           //---------------
                           IF "SysTick1s" THEN
                               #i   :=  #i + 1;
                           END_IF;
                           //increase step counter
                           //---------------------
                           IF (#i > 120) THEN
                               #step    :=  #step + 10;
                               #i       :=  0;
                           END_IF;
                       END_IF;
                   END_IF;

               20: //close valve V1 and wait 1sec
                   //----------------------------
                   "AC".SET_CTL_VALVE_POS    :=  0.0;      //close pressure control valve

                   IF NOT "LT".V1_OPEN THEN 
                       //count wait time
                       //---------------
                       IF "SysTick100ms" THEN
                           #i   :=  #i + 1;
                       END_IF;
                       //increase step counter
                       //---------------------
                       IF (#i > 10) THEN
                           #step    :=  #step + 10;
                           #i       :=  0;
                       END_IF;
                   END_IF;

               30: //open V22 for for configured blowback duration
                   //---------------------------------------------
                   IF NOT #fill_up_sto_tank THEN    //fill up already done, set V22 open request
                       "DC".V22_OP   :=  TRUE;
                   END_IF;
                   //blowback
                   //--------
                   IF "PDO".V22  THEN 
                       //count blowbacks
                       //---------------
                       IF ((#i > "CNF".V22_OP_TME) OR ("DIS".ACT_PRS_AR_VSL <= "CNF".MIN_PRS_AR_VSL)) THEN
                           #count   :=  #count + 1;
                           #step    :=  #step + 10;
                           #i       :=  0;
                       ELSE
                           //increase open time
                           //------------------
                           #i   :=  #i + "SY".OB1_PREV_CYCLE;
                       END_IF;
                   END_IF;

               40: //close V22
                   //---------
                   "DC".V22_OP   :=  FALSE;
                   //valve closed
                   //------------
                   IF NOT "PDO".V22 THEN
                       //check amount of pulses after two seconds wait time
                       //--------------------------------------------------
                       IF (#i > 20) THEN
                           IF (#count < "CNF".AMT_OF_V22_BB) THEN 
                               #step    :=  #step + 10;
                           ELSE
                               #step    :=  #step + 30;
                           END_IF;
                           #i   :=  0;
                       ELSIF "SysTick100ms" THEN
                           #i := #i + 1;
                       END_IF;
                   END_IF; 


               50: //request fill up of gas storage tank
                   //-----------------------------------
                   #fill_up_sto_tank    :=  true;
                   #step                :=  #step + 10;
                   #i                   :=  0;

               60: //wait untill fill up of storage tank is done
                   //-------------------------------------------
                   IF NOT #fill_up_sto_tank THEN
                       //wait two seconds after tank filled
                       //----------------------------------
                       IF (#i > 20) THEN
                           #step    :=  #step - 30;
                           #i       :=  0;
                       ELSIF "SysTick100ms" THEN
                           #i := #i + 1;
                       END_IF;
                   END_IF;   

               70: //wait 10 seconds
                   //---------------
                   "DC".P1_ON    :=  FALSE;      //stop vacuum pump
                   //increase step counter
                   //---------------------
                   IF (#i > 10) THEN   
                       #step    :=  #step + 10;
                       #i       :=  0;
                   //count wait time
                   //----------------
                   ELSIF "SysTick1s" THEN
                       #i   :=  #i + 1;
                   END_IF;


               80: //V20 open; flush filter with air 
                   //--------------------------
                   "DC".V20_OP   :=  TRUE;

                   IF "PDO".V20  THEN            
                       IF "PDI".FIL_APS AND "PDI".FCH_APS THEN
                           #step    :=  #step + 10;
                       END_IF;
                       IF "LT".V7_OPEN THEN
                          "DC".V4_OP := NOT "DV".APS_FCH_DELAYED;
                       ELSE   
                          "DC".V6_OP := NOT "DV".APS_FCH_DELAYED;
                          "DC".V4_OP := NOT "DV".APS_GCH_DELAYED;
                          IF "PDO".V6 THEN
                             "AC".SET_GAS_1_FLW := 50.0;
                          ELSE
                             "AC".SET_GAS_1_FLW := 0.0;
                          END_IF;
                      END_IF;           
                   END_IF;       


               90: //close air inlet valve and reset gas flow 1 set point
                   //----------------------------------------------------    
                   "DC".V20_OP           :=  FALSE;
                   "AC".SET_GAS_1_FLW    :=  0.0;

                   //count wait time
                   //---------------
                   IF "SysTick100ms" THEN
                       #i   :=  #i + 1;
                   END_IF;
                   //increase step counter
                   //---------------------
                   IF (#i > 5) THEN
                       #step    :=  #step + 10;
                       #i       :=  0;
                   END_IF;

              100: //finish filter flushing sequence
                   //-------------------------------             
                   #req_fil_cln             :=  false;
                   #run_fil_cln             :=  false;
                   "DV".SI_FIL_FSH_REQ       :=  FALSE;
                   "LT".SI_FIL_FSH_SEQ_ON    :=  FALSE;


              110: //abort filter flushing - stop pump and close valves
                   //--------------------------------------------------
                   "DC".V20_OP               :=  FALSE;      //close air inlet valve
                   "DC".V22_OP               :=  FALSE;      //close Ar inlet valve filter
                   "DV".V25_OP               :=  FALSE;      //close Ar inlet storage tank
                   #fill_up_sto_tank        :=  false;      //reset fill up request storage tank
                   "DC".V19_OP               :=  FALSE;      //close dust outlet valve filter
                   "DC".P1_ON                :=  FALSE;      //stop vacuum pump
                   "AC".SET_CTL_VALVE_POS    :=  0.0;        //close pressure control valve

                   //count wait time
                   //---------------
                   IF "SysTick100ms" THEN
                       #i   :=  #i + 1;
                   END_IF;
                   //increase step counter
                   //---------------------
                   IF (#i > 20) THEN
                       #step    :=  #step + 10;
                       #i       :=  0;
                   END_IF;

              120: //abort filter flushing - switch off filter flushing sequence and set alarm message
                   //---------------------------------------------------------------------------------
                   #req_fil_cln             :=  false;
                   #run_fil_cln             :=  false;
                   "FLT".SI_FIL_REG_ENB      :=  TRUE;
                   "LT".SI_FIL_FSH_SEQ_ON    :=  FALSE;
           END_CASE;

       ELSE
           #step    :=  0;              //reset step counter

       END_IF;

       //reset global aux flag regeneration sequence is active
       //-----------------------------------------------------
       IF NOT #run_fil_cln THEN 
           "DV".SI_FIL_FSH_SEQ_ON    :=  FALSE;
       END_IF;
END_FUNCTION_BLOCK

FUNCTION_BLOCK "BM_CDP"   // FB89, SCL
{ S7_Optimized_Access := 'FALSE' }
VERSION : 0.0
// --------------------------------------------------------------------------------
//     program     :    BM_CDP
//     description :    
//     name        :    G. Eibelsh鋟ser
//     date        :    16.12.2008
//     
//     revision    :   
//     name        :   
//     date        :  
//     
//     Info        :   AUX_FLAGS - 0   -   new carrier ID
//                                 1   -   Ingot ID transfered to PLC
//                                 2   -   Growth process is running
//                                 3   -   Teilkristall removal
//                                 4   -   Sputnik removal
//                                 5   -   Crucible breakage
//                                 6   -   Melt back
//                                 7   -   Melting of Si-rods
//                                 8   -   puller failure
//                                 9   -   emergency situation
//                                10   -   other reasons for manual mode
//                                11   -   spare
//                                12   -   spare
//                                13   -   spare
//                                14   -   spare
//                                15   -   spare
//                                16   -   spare
//                                17   -   spare
//                                18   -   spare
//                                19   -   spare
//                                20   -   spare
//                                21   -   spare
//                                22   -   spare
//                                23   -   spare
//                                24   -   spare
//                                25   -   spare
//                                26   -   spare
//                                27   -   spare
//                                28   -   spare
//                                29   -   spare
//                                30   -   spare
//                                31   -   spare
// 
//                     (c)CGS
//     --------------------------------------------------------------------------------
   VAR
      FLT : Array[1..580] of Bool;
      FLT_STOR : Array[1..580] of Bool;
      i : Int;
      RETVAL : Int;
      OLD_XT_LEN_MM : Real;
   END_VAR
BEGIN


   (*
       //ID-transfer PLC <> CDP in machine state service
       //-----------------------------------------------
       IF (STA.ACT_STATE = APC.STATE_SERV)  THEN           //state service is activated

           //set default values
           //------------------
           IF NOT init_aux_flag_srv   THEN
               STA.AUX_FLAGS       :=  2#0000_0000_0000_0000_0000_0000_0000_0000;

               //reset global strings byte by byte - delete function FC4 not working
               //-------------------------------------------------------------------
               FOR address:= 656 TO 665 DO                 //reset 10 bytes of carrier ID
                   DB204.DBB[address]    :=  B#16#00;
               END_FOR;

               FOR address:= 244 TO 443 DO                 //reset 200 bytes of ingot ID
                   DB204.DBB[address]    :=  B#16#00;
               END_FOR;

               new_carrier_id      :=  false;
               ingot_id_rcv        :=  false;
               set_carrier_id_done :=  false;

               LT.ENB_LOADING      :=  FALSE;          //disable crucible loading of puller
               LT.EDIT_INGOT_ID    :=  FALSE;

               init_aux_flag_srv   :=  true;

           END_IF;

           //enable editing of carrier ID
           //----------------------------
           IF NOT new_carrier_id AND NOT ingot_id_rcv THEN 
               LT.EDIT_CARRIER_ID  :=  TRUE;
               STA.AUX_FLAGS       :=  2#0000_0000_0000_0000_0000_0000_0000_0000;
           ELSE
               LT.EDIT_CARRIER_ID  :=  FALSE;
           END_IF;

           //carrier ID
           //----------
           IF KYD.NEW_CARRIER_ID AND NOT new_carrier_id AND NOT ingot_id_rcv  THEN //new carrier ID is edited
               LT.EDIT_INGOT_ID        :=  FALSE;
               new_carrier_id          :=  true;
           END_IF;

           //delay carrier ID flag
           //---------------------
           set_carrier_id  := SysOndelay(  DIN     := new_carrier_id,
                                           SetTime := dly_set_carrier_id,      // setp. time
                                           ActTime := set_carrier_id_dly,      // act. time
                                           Tick    := SysTick100ms);           // timebase (100ms)

           //delay carrier ID flag
           //---------------------
           IF set_carrier_id AND NOT set_carrier_id_done THEN 
               STA.AUX_FLAGS           :=  STA.AUX_FLAGS OR 2#0000_0000_0000_0000_0000_0000_0000_0001;
               set_carrier_id_done     :=  true;
           END_IF;

           //response from CDP
           //-----------------
           IF NOT LT.EDIT_INGOT_ID THEN                                   //manual editing of ingot ID disabled
               IF (STA.AUX_FLAGS AND 2#0000_0000_0000_0000_0000_0000_0000_0011) = 2#0000_0000_0000_0000_0000_0000_0000_0011 THEN    //ingot ID has been generated
                   STA.ACT_INGOT_ID    :=  STA.AUX_INFO;
                   ingot_id_rcv        :=  true;

               END_IF;
           END_IF;  

           //reset flags 
           //-----------
           IF (reset_aux_flags OR (KYD.INGOT_ID_EDIT AND LT.EDIT_INGOT_ID)) THEN
               STA.AUX_FLAGS   :=  STA.AUX_FLAGS AND 2#1111_1111_1111_1111_1111_1111_1111_1100;  
               ingot_id_rcv    :=  false;      //reset flag and enable new editing of carrier ID

               //carrier ID refused from MES - reset flag
               //----------------------------------------
               IF (STA.ACT_INGOT_ID = carrier_id_refused) THEN                                          
                   new_carrier_id      :=  false;
                   set_carrier_id_done :=  false;
                   LT.ENB_LOADING      :=  FALSE;      //disable crucible loading of puller
               ELSE
                   LT.ENB_LOADING      :=  TRUE;       //enable crucible loading of puller
               END_IF;

           END_IF;

           //reset aux flags
           //---------------
           init_aux_flag_prc   :=  false;

       //machine state process
       //---------------------
       ELSIF (STA.ACT_STATE = APC.STATE_RUN)  THEN         //state process is activated
           //set process is running flag
           //---------------------------





           IF NOT init_aux_flag_prc  THEN 
               STA.AUX_FLAGS       :=  2#0000_0000_0000_0000_0000_0000_0000_0100;
               init_aux_flag_prc   :=  true;
           END_IF;

           //new ingot ID after crystal part removal
           //---------------------------------------
           IF (STA.MAN_SEL_REAS = 3) OR (APC.STATUS = APC.REMOVAL) THEN

               //check pressure status in gate chamber
               //-------------------------------------
               IF act_cgt_prs_sta AND NOT DV.APS_GCH_DELAYED THEN  //switched from atmosphere to vacuum?
                   new_ingot_id_req    :=  true;
               END_IF;

               //request new ingot ID from CDP
               //-----------------------------
               IF new_ingot_id_req THEN 
                   FOR address:= 244 TO 443 DO                 //reset 200 bytes of ingot ID
                       DB204.DBB[address]    :=  B#16#00;
                   END_FOR;

                   STA.AUX_FLAGS       :=  STA.AUX_FLAGS OR 2#0000_0000_0000_0000_0000_1000_0000_0000;
                   new_ingot_id_is_req :=  true;   
                   new_ingot_id_req    :=  false;
               END_IF;
           ELSE 
               new_ingot_id_req    :=  false;

           END_IF;

           //response from CDP
           //-----------------
           IF new_ingot_id_is_req THEN 
               IF (STA.AUX_FLAGS AND 2#0000_0000_0000_0000_0000_0000_0000_0010) = 2#0000_0000_0000_0000_0000_0000_0000_0010 THEN    //ingot ID has been generated
                   STA.ACT_INGOT_ID    :=  STA.AUX_INFO;
                   ingot_id_rcv        :=  true;
               END_IF;
           END_IF;

           //reset flags 
           //-----------
           IF (reset_aux_flags OR (KYD.INGOT_ID_EDIT AND LT.EDIT_INGOT_ID)) THEN
               STA.AUX_FLAGS       :=  STA.AUX_FLAGS AND 2#1111_1111_1111_1111_1111_0111_1111_1100;  
               ingot_id_rcv        :=  false;      //reset flag and enable new editing of carrier ID
               new_ingot_id_is_req :=  false;
           END_IF;

           //reset aux flag loading state
           //----------------------------
           init_aux_flag_srv   :=  false;

       END_IF;

       //delay reset of aux flags after ingot ID received
       //------------------------------------------------
       reset_aux_flags :=  SysOndelay( DIN     := ingot_id_rcv,
                                       SetTime := dly_reset,           // setp. time
                                       ActTime := reset_dly,           // act. time
                                       Tick    := SysTick100ms);       // timebase (100ms)

       //alarm message timeout ingot ID
       //------------------------------
       ingot_id_time_out   :=  SysOndelay( DIN     := new_carrier_id OR new_ingot_id_is_req,
                                           SetTime := STA.INGOT_ID_TIMEOUT,    // setp. time
                                           ActTime := time_out_dly,            // act. time
                                           Tick    := SysTick1s);              // timebase (1s)

       //enable manual editing of ingot ID - communication with CDP failed
       //-----------------------------------------------------------------
       IF ingot_id_time_out THEN
           LT.EDIT_INGOT_ID    :=  TRUE;
           new_carrier_id      :=  false;
           set_carrier_id_done :=  false;
           new_ingot_id_is_req :=  false;
       END_IF;

       //additional cases for manual mode
       //--------------------------------
       IF APC.AUTOMATIC    THEN 
           //reset manual selection after automatic is activated again
           //---------------------------------------------------------
           IF init_stat_reset  THEN
               STA.MAN_SEL_REAS        :=  0;
               STA.AUX_FLAGS           :=  STA.AUX_FLAGS AND 2#1111_1111_1111_1111_1111_1000_0000_0111;
               init_stat_reset         :=  false;

           END_IF;

           //manual selection before switching from automatic to manual
           //----------------------------------------------------------
           IF (STA.MAN_SEL_REAS =  1)   THEN           //remelt after dislocations
               STA.AUX_FLAGS   :=  STA.AUX_FLAGS OR 2#0000_0000_0000_0000_0000_0000_0100_0000;
           ELSIF (STA.MAN_SEL_REAS =  2) THEN          //melting of Si rods
               STA.AUX_FLAGS   :=  STA.AUX_FLAGS OR 2#0000_0000_0000_0000_0000_0000_1000_0000;
           ELSIF (STA.MAN_SEL_REAS =  3) THEN          //remove of crystal part
               STA.AUX_FLAGS   :=  STA.AUX_FLAGS OR 2#0000_0000_0000_0000_0000_0000_0000_1000;
           ELSIF (STA.MAN_SEL_REAS =  4) THEN          //remove of sputnik
               STA.AUX_FLAGS   :=  STA.AUX_FLAGS OR 2#0000_0000_0000_0000_0000_0000_0001_0000;
           ELSIF (STA.MAN_SEL_REAS =  5) THEN           //crucible leakage
               STA.AUX_FLAGS   :=  STA.AUX_FLAGS OR 2#0000_0000_0000_0000_0000_0000_0010_0000;
           ELSIF (STA.MAN_SEL_REAS =  6) THEN           //puller failure
               STA.AUX_FLAGS   :=  STA.AUX_FLAGS OR 2#0000_0000_0000_0000_0000_0001_0000_0000;
           ELSIF (STA.MAN_SEL_REAS =  7) THEN          //emergency situation
               STA.AUX_FLAGS   :=  STA.AUX_FLAGS OR 2#0000_0000_0000_0000_0000_0010_0000_0000;
           ELSIF (STA.MAN_SEL_REAS =  8) THEN          //other reason
               STA.AUX_FLAGS   :=  STA.AUX_FLAGS OR 2#0000_0000_0000_0000_0000_0100_0000_0000;
           END_IF;

       ELSE 
           init_stat_reset :=  true;       //reset aux flag

       END_IF;

       //free editable comment
       //---------------------
       IF (STA.AUX_FLAGS AND 2#0000_0000_0000_0000_0001_0000_0000_0000) = 2#0000_0000_0000_0000_0001_0000_0000_0000 THEN    //ingot ID has been generated
           IF (i > 50) THEN
               //reset comment
               //-------------
               FOR address:= 870 TO 1123 DO                 //reset 254 bytes of free editable comment
                   DB204.DBB[address]    :=  B#16#00;
               END_FOR;

               STA.AUX_FLAGS   :=  (STA.AUX_FLAGS AND 2#1111_1111_1111_1111_1110_1111_1111_1111);  //reset bit 12 of aux flag
           ELSE
               i := i + 1;                                                                         //increment delay counter
           END_IF;
       ELSE        
           i   :=  0;                                                                              //reset delay counter
       END_IF;

       //machine state according Semi E10
       //--------------------------------
       IF (STA.ACT_STATE = APC.STATE_MAINTENANCE)  THEN    
           STA.SEMI_E10_STATE  :=  5;                          //SD - scheduled down time
       ELSIF (STA.ACT_STATE = APC.STATE_ENGINEERING) OR (STA.ACT_STATE = APC.STATE_VAC_TEST) THEN
           STA.SEMI_E10_STATE  :=  4;                          //EN - engineering time
       ELSIF (STA.ACT_STATE = APC.STATE_STD_BY)  THEN
           STA.SEMI_E10_STATE  :=  3;                          //SB - standby time
       ELSIF LT.MA_NOT_AVL THEN
           STA.SEMI_E10_STATE  :=  6;                          //UD - unscheduled down time
       ELSE
           STA.SEMI_E10_STATE  :=  2;                          //PR - productive time
       END_IF;

       //store pressure status in gate chamber every 100ms
       //-------------------------------------------------
       IF SysTick100ms THEN 
           act_cgt_prs_sta :=  DV.APS_GCH_DELAYED;
       END_IF;

       *)

      // SEND_MES.Header    :=  STA.Header;

       IF ("SysTick1s" AND ("APC".STATUS<>"APC".BODY)) OR 
          ("APC".STATUS="APC".BODY) AND ("DIS".ACT_XT_LEN_MM-#OLD_XT_LEN_MM)>1.0 THEN

          #OLD_XT_LEN_MM           := "DIS".ACT_XT_LEN_MM;

         // SEND_MES.MachineNo      :=  STA.MachineNo;
          "SEND_MES".MachineStatus  :=  "STA".ACT_STATE;
          "SEND_MES".ACT_PROCESS    :=  "STA".ACT_PROCESS;
         // SEND_MES.Timestamp      :=  STA.ACT_PC_TIME;
          "SEND_MES".User_Name      BLKMOV  "STA".USER_NAME;
          "SEND_MES".ACT_RCP_NAME   BLKMOV  "STA".ACT_RCP_NAME;
          "SEND_MES".ACT_INGOT_ID   BLKMOV  "STA".ACT_INGOT_ID;
          "SEND_MES".ACT_CHARGE_ID  BLKMOV  "STA".ACT_CHARGE_ID;
          "SEND_MES".ACT_CRU_ID     BLKMOV  "STA".ACT_CRU_ID;

          "SEND_MES".ACT_XT_SPD     :=  "DIS".ACT_XT_SPD;
          "SEND_MES".ACT_XT_ROT     :=  "DIS".ACT_XT_ROT;
          "SEND_MES".ACT_XT_POS     :=  "DIS".ACT_XT_POS;
          "SEND_MES".ACT_CR_SPD     :=  "DIS".ACT_CR_SPD;
          "SEND_MES".ACT_CR_ROT     :=  "DIS".ACT_CR_ROT;
          "SEND_MES".ACT_CR_POS     :=  "DIS".ACT_CR_POS;
          "SEND_MES".ACT_HTR_1_PWR  :=  "DIS".ACT_HTR_1_PWR;
          "SEND_MES".ACT_HTR_1_TMP  :=  "DIS".ACT_HTR_1_TMP;
          "SEND_MES".ACT_HTR_2_PWR  :=  "DIS".ACT_HTR_2_PWR;
          "SEND_MES".ACT_MAG_1_CUR  :=  "DIS".ACT_MAG_1_CUR;
          "SEND_MES".ACT_MAG_2_CUR  :=  "DIS".ACT_MAG_2_CUR;
          "SEND_MES".ACT_GAS_1_FLW  :=  "DIS".ACT_GAS_1_FLW;
          "SEND_MES".ACT_GAS_2_FLW  :=  "DIS".ACT_GAS_2_FLW;
          "SEND_MES".ACT_TOT_XT_LGH :=  "DIS".ACT_TOT_XT_LGH;
          "SEND_MES".ACT_PRS_CLF    :=  "DIS".ACT_PRS_CLF;
          "SEND_MES".ACT_PRS_CGT    :=  "DIS".ACT_PRS_CGT;
          "SEND_MES".ACT_XT_DIA     :=  "DIS".ACT_XT_DIA;
          "SEND_MES".ACT_XT_LEN_MM  :=  "DIS".ACT_XT_LEN_MM;
          "SEND_MES".CHARGE_WGT     :=  "PAR_MAIN".CH_SILICON_CHARGE;
          "SEND_MES".CRU_QRZ_WALL_THICKN :=  "PAR_MAIN".CH_QRZ_WALL_THICKN;
          "SEND_MES".CRU_QRZ_BOT_THICKN  :=  "PAR_MAIN".CH_QRZ_BOTTOM_THICKN;
          "SEND_MES".CRU_QRZ_TRANS_RAD   :=  "PAR_MAIN".CH_GRAPH_TRANS_RAD;
          "SEND_MES".CRU_GRAPH_BOT_RAD   :=  "PAR_MAIN".CH_GRAPH_BOTTOM_RAD;
          "SEND_MES".CRU_GRAPH_INNER_DIA :=  "PAR_MAIN".CH_GRAPH_INNER_DIA;
       END_IF; 


       // Write fault history list
       //-----------------------------------------------
       IF "SysTick500ms" THEN
          "FLT_BLKMOV"();
          FOR #i := 1 TO 580 DO
              IF #FLT[#i] AND NOT #FLT_STOR[#i] THEN           // Check if a new fault is active
                 "SEND_MES".FAULT[10] := "SEND_MES".FAULT[9];
                 "SEND_MES".FAULT[9]  := "SEND_MES".FAULT[8];
                 "SEND_MES".FAULT[8]  := "SEND_MES".FAULT[7];
                 "SEND_MES".FAULT[7]  := "SEND_MES".FAULT[6];
                 "SEND_MES".FAULT[6]  := "SEND_MES".FAULT[5];
                 "SEND_MES".FAULT[5]  := "SEND_MES".FAULT[4];
                 "SEND_MES".FAULT[4]  := "SEND_MES".FAULT[3];
                 "SEND_MES".FAULT[3]  := "SEND_MES".FAULT[2];
                 "SEND_MES".FAULT[2]  := "SEND_MES".FAULT[1];
                 "SEND_MES".FAULT[1]  := #i;                  // Write ring buffer and set the new detected fault on top(1) of the list
                 #FLT_STOR[#i]        := #FLT[#i];             // And store the information to the stored aera 
               END_IF;
              IF NOT #FLT[#i] AND #FLT_STOR[#i] THEN
                 #FLT_STOR[#i]        := #FLT[#i];             // reset gone faults in the stored aera   
              END_IF;
          END_FOR;
       END_IF;
END_FUNCTION_BLOCK

FUNCTION_BLOCK "BM_XT_ORB_DET"   // FB92, SCL
{ S7_Optimized_Access := 'FALSE' }
VERSION : 0.0
// --------------------------------------------------------------------------------
//     program     :    BM_XT_ORB_DET
//     description :    crystal orbiting detection       
//     name        :    G. Eibelsh鋟ser
//     date        :    01.10.2009
// 
//     revision    :
//     name        :
//     date        :    
//                     (c)PVATepla AG
//     --------------------------------------------------------------------------------
   VAR
      enb_orb_mon : Bool;
      orb_calc_done : Bool;
      msr_per_rot : Int;
      count_msr : Int;
      set_flt : Int;
      reset_flt : Int;
      xt_orb_mm : Real;
      up_lim_xt_orb : Real;
      rst_lim_xt_orb : Real;
      ctr_x_val : Array[1..300] of Real;
      min_val_ctr_x_pos : Real;
      max_val_ctr_x_pos : Real;
   END_VAR
BEGIN


       //activate crystal orbiting monitoring
       //------------------------------------
       #enb_orb_mon :=  ((("APC".STATUS = "APC".NECK) AND ("PAR_MAIN".MCONST_XT_ORB_LIM_NE > 0.0)) OR 
                       (("APC".STATUS = "APC".SHOULDER) AND ("PAR_MAIN".MCONST_XT_ORB_LIM_SH > 0.0)) OR 
                       (("APC".STATUS = "APC".BODY) AND ("PAR_MAIN".MCONST_XT_ORB_LIM_BY > 0.0))) AND 
                       ("DIS".SET_XT_ROT >= 2.0)     AND 
                       ("AV".ACT_DVT_PRD_NO = 2.0)   AND
                       "LT".CAM_ISP_ON;

       //crystal orbiting is activated
       //-----------------------------                          
       IF #enb_orb_mon  THEN

           //reset calculation done flag
           //---------------------------
           #orb_calc_done   :=  false;            

           //calculate amount of diameter measurements on one rotation of crystal 
           //--------------------------------------------------------------------
           #msr_per_rot := REAL_TO_INT(60000 / "CNF".IMG_AQI_TRG / "DIS".SET_XT_ROT);      //60000ms = 1 min, max. 300 values in array

           //read sensor center coordinate
           //-----------------------------   
           IF "DV".NEW_MSR_TEL_RECV THEN                              //new measurement telegram received
               #count_msr               := #count_msr + 1;           //increase counter variable after each measurement
               #ctr_x_val[#count_msr]    := "AV".ACT_PRD_2_CTR_X;      //store center position in array variable
           END_IF;

           //evaluate measurement points   
           //---------------------------
           IF (#count_msr >= #msr_per_rot) THEN

               //call min max detection
               //----------------------
               "CM_MIN_MAX"( record      := #ctr_x_val,
                           amt_of_val  := #msr_per_rot,
                           min_value   := #min_val_ctr_x_pos, 
                           max_value   := #max_val_ctr_x_pos);

